# B&R Automation Studio project Embraco_LinkaNaOdlievanieRotorov_DokoncovaciaStanica_Rev2 (part 2)

#### Axis.c - Axis control
```c
 /********************************************************************
  * COPYRIGHT -- Bernecker + Rainer
  ********************************************************************
  * Author: Milan Jun
  * Created: May 28, 2014
  ********************************************************************/

#include <bur/plctypes.h>
#ifdef __cplusplus
	extern "C"
	{
#endif

#include "AxisLib.h"

#ifdef __cplusplus
	};
#endif

#define TRUE	1      /* Allways true */
#define FALSE 	0      /* Allways false */
#define DELAY   100    /* Delay time, it is dependence on cycle time */

/* Disabled all commands and executes */
void AxisDisableCmd (struct Axis* inst)
{

	/* RESET ALL FB EXECUTE/ENABLE INPUT */
	inst->internal.MC_Power_0.Enable = FALSE;
	inst->internal.MC_Home_0.Execute = FALSE;
	inst->internal.MC_Halt_0.Execute = FALSE;
	inst->internal.MC_Stop_0.Execute = FALSE;
	inst->internal.MC_MoveAbsolute_0.Execute = FALSE;
	inst->internal.MC_MoveAdditive_0.Execute = FALSE;
	inst->internal.MC_MoveVelocity_0.Execute = FALSE;
	inst->internal.MC_TorqueControl_0.Execute = FALSE;
	inst->internal.MC_BR_VelocityControl_0.Enable = FALSE;

	/* RESET USER COMMANDS */
	inst->cmd.home = FALSE;
	inst->cmd.halt = FALSE;
	inst->cmd.stop = FALSE;
	inst->cmd.moveAbsolute = FALSE;
	inst->cmd.moveAdditive = FALSE;
	inst->cmd.moveVelocity = FALSE;
	inst->cmd.moveVelocityControl = FALSE;
	inst->cmd.moveTorqueControl = FALSE;
	inst->cmd.moveJogPos = FALSE;
	inst->cmd.moveJogNeg = FALSE;
	inst->cmd.moveTorqueControl = FALSE;
	// inst->cmd.autoInicialization = FALSE;
	inst->errorID = FALSE;

}

/* Disabled all commands and executes */
void AxisAutoInicialization (struct Axis* inst)
{
 /* *************************************************************** *
 * ************** AUTO INICIALIZATION ENABLED ******************** *
 * *************************************************************** */
	switch (inst->internal.InitStep)
	{

		/* Init state */
		case STATE_INIT:
			inst->cmd.errorAck = FALSE;
			inst->internal.switch1 = FALSE;
			inst->internal.switch2 = FALSE;
			inst->internal.TimeCheck = 0;
			inst->internal.InitStep = STATE_WATCH;
			break;

		/* Wait for action, homing, power, error acknowledge */
		case STATE_WATCH:

			//   if ( (inst->status.DriveStatus.NetworkInit == TRUE) &&
			//   (inst->status.DriveStatus.HomingOk == FALSE) &&
			//   (inst->status.DriveStatus.ControllerStatus == TRUE) &&
			//   (inst->state.ErrorStop == FALSE) &&
			//			(inst->status.DriveStatus.AxisError == FALSE)	)
			//   {
			//    inst->internal.InitStep = STATE_HOME;
			//   }

			if ((inst->status.DriveStatus.NetworkInit == TRUE) &&
				(inst->status.DriveStatus.ControllerReady == TRUE) &&
				(inst->status.DriveStatus.ControllerStatus == FALSE) &&
				(inst->state.ErrorStop == FALSE) &&
				(inst->status.DriveStatus.AxisError == FALSE)	)
			{
				inst->internal.InitStep = STATE_SWITCHON;
			}

			if ((inst->status.DriveStatus.NetworkInit == TRUE) && ((inst->state.ErrorStop == TRUE) || (inst->status.DriveStatus.AxisError == TRUE) || (inst->errorID!=0)))
			{
				inst->internal.InitStep = STATE_ERROR_HANDLE;
			}
			break;

		/* State: homing */
		case STATE_HOME:

			if (inst->internal.switch1 == FALSE)
			{
				inst->cmd.home = TRUE;
				inst->internal.switch1 = TRUE;
			}

			if (inst->status.DriveStatus.HomingOk == TRUE)
			{
			inst->internal.InitStep = STATE_INIT;
			}

			inst->internal.TimeCheck = inst->internal.TimeCheck + 1;

			if (inst->internal.TimeCheck == DELAY)
			{
				inst->internal.InitStep = STATE_INIT;
				inst->internal.TimeCheck = 0;
			}
			break;

		/* State: switching on */
		case STATE_SWITCHON:

			if (inst->internal.switch1 == FALSE)
			{
				inst->cmd.power = TRUE;
				inst->internal.switch1 = TRUE;
			}

			if (inst->status.DriveStatus.ControllerStatus == TRUE)
			{
			inst->internal.InitStep = STATE_INIT;
			}

			inst->internal.TimeCheck = inst->internal.TimeCheck + 1;

			if (inst->internal.TimeCheck == DELAY)
			{
				inst->internal.InitStep = STATE_INIT;
				inst->internal.TimeCheck = 0;
			}
			break;

		/* State: automatic error acknowledge */
		case STATE_ERROR_HANDLE:

			inst->internal.errorOld = inst->errorID;

			if (inst->internal.switch1 == FALSE)
			{
			//inst->cmd.power = FALSE;
			inst->internal.switch1 = TRUE;
			}

			if ((inst->internal.switch1 == TRUE) && (inst->internal.switch2 == FALSE))
			{
			inst->cmd.errorAck = TRUE;
			inst->internal.switch2 = TRUE;
			}

			if (inst->internal.errorOld != inst->errorID)
			{
				inst->internal.errorOld = FALSE;
				inst->cmd.errorAck = FALSE;
				inst->internal.InitStep = STATE_INIT;
			}

			inst->internal.TimeCheck = inst->internal.TimeCheck + 1;

			if (inst->internal.TimeCheck == DELAY)
			{
				inst->internal.InitStep = STATE_INIT;
				inst->internal.TimeCheck = 0;
			}
			break;

	} /* END AutoInicialization enabled */

} /* END AutoInicialization disabled */

/* *************************************************************** *
 * ************************ AXIS CONTROL ************************* *
 * *************************************************************** */
void Axis(struct Axis* inst)
{

	/* Function Block is Enabled */
	if (inst->enable == TRUE){

		/* Function block active, when network iniciaization is true */
		if ( inst->status.DriveStatus.NetworkInit == TRUE )
		{
			inst->busy = FALSE;
			inst->active = TRUE;
		}
		else
		{
			inst->busy = TRUE;
			inst->active = FALSE;
		}

  /* *************************************************************** *
   * ************** AUTO INICIALIZATION DISABLED ******************* *
   * *************************************************************** */

		if ( inst->cmd.autoInicialization == FALSE )
		{
			inst->internal.switch1 = FALSE;
			inst->internal.TimeCheck = 0;
			inst->internal.InitStep = STATE_INIT;
		}
		else AxisAutoInicialization(inst);

  /* ******************** *
   * MC READ DRIVE STATUS *
   * ******************** */
		inst->internal.MC_BR_ReadDriveStatus_0.Enable = !inst->internal.MC_BR_ReadDriveStatus_0.Error;
		inst->internal.MC_BR_ReadDriveStatus_0.Axis = inst->par.axis;
		inst->internal.MC_BR_ReadDriveStatus_0.AdrDriveStatus = (UDINT)&inst->status.DriveStatus;

  /* ************** *
   * MC READ STATUS
   * ************** */
		inst->internal.MC_ReadStatus_0.Enable = !inst->internal.MC_ReadStatus_0.Error;
		inst->internal.MC_ReadStatus_0.Axis = inst->par.axis;

		/* MC READ ACTUAL POSITION */
		inst->internal.MC_ReadActualPosition_0.Enable = (!inst->internal.MC_ReadActualPosition_0.Error);
		inst->internal.MC_ReadActualPosition_0.Axis = inst->par.axis;

		if (inst->internal.MC_ReadActualPosition_0.Valid == TRUE)
		{
			inst->status.ActPosition = inst->internal.MC_ReadActualPosition_0.Position;
		}

		/* MC READ ACTUAL VELOCITY */
		inst->internal.MC_ReadActualVelocity_0.Enable = (!inst->internal.MC_ReadActualVelocity_0.Error);
		inst->internal.MC_ReadActualVelocity_0.Axis = inst->par.axis;

		if(inst->internal.MC_ReadActualVelocity_0.Valid == TRUE)
		{
			inst->status.ActVelocity = inst->internal.MC_ReadActualVelocity_0.Velocity;
		}

		/* MC READ ACTUAL TORQUE */
		inst->internal.MC_ReadActualTorque_0.Enable = (!inst->internal.MC_ReadActualTorque_0.Error);
		inst->internal.MC_ReadActualTorque_0.Axis = inst->par.axis;

		if(inst->internal.MC_ReadActualTorque_0.Valid == TRUE)
		{
			inst->status.ActTorque = inst->internal.MC_ReadActualTorque_0.Torque;
		}

		/* MC READ AXIS ERROR */
		inst->internal.MC_ReadAxisError_0.Enable = !inst->internal.MC_ReadAxisError_0.Error;
		inst->internal.MC_ReadAxisError_0.Axis = inst->par.axis;
		inst->internal.MC_ReadAxisError_0.DataAddress = (UDINT)&(inst->errorText);
		inst->internal.MC_ReadAxisError_0.DataLength = sizeof(inst->errorText);
		brsstrcpy((void*)&inst->internal.MC_ReadAxisError_0.DataObjectName, "acp10etxen");

		/* CHECK FOR GENERAL AXIS ERROR */
		if ((inst->internal.MC_ReadAxisError_0.AxisErrorID != FALSE) &&
			(inst->internal.MC_ReadAxisError_0.Valid == TRUE))
		{
			inst->internal.AxisStep = AXISSTATE_ERROR_AXIS;
		}

		/* Main Cyclic Part */

		if ( inst->cmd.power == FALSE )
		{
			inst->internal.MC_Power_0.Enable = FALSE;
			inst->internal.AxisStep = AXISSTATE_WAIT;
		}

		/* State machine for axis */
		switch (inst->internal.AxisStep)
		{
			/* STATE WAIT FOR POWERON */
			case AXISSTATE_WAIT:

				/* WAIT FOR POWERON COMMAND */
				if (inst->cmd.power == TRUE) {
					inst->internal.AxisStep = AXISSTATE_POWER_ON;
				}
				else {
					inst->internal.MC_Power_0.Enable = FALSE;
				}

				AxisDisableCmd(inst);

				break;

   /* *************************************************************** *
    * ************************ STATE POWER ON *********************** *
    * *************************************************************** */
			case AXISSTATE_POWER_ON:
				inst->internal.MC_Power_0.Axis = inst->par.axis;
				inst->internal.MC_Power_0.Enable = TRUE;

				/* Check staus ok */
				if (inst->internal.MC_Power_0.Status == TRUE) {
					inst->internal.AxisStep = AXISSTATE_READY;
				}
				/* Check a power error, then go to error state */
				if (inst->internal.MC_Power_0.Error == TRUE) {
					inst->errorID = inst->internal.MC_Power_0.ErrorID;
					inst->internal.AxisStep = AXISSTATE_ERROR;
				}
				break;
			/* ************************************************************** */

			/* ************************************************************** *
			* ************************* STATE READY ************************* *
			* *************************************************************** */
			case AXISSTATE_READY:
				if (inst->cmd.home == TRUE) {
					inst->internal.AxisStep = AXISSTATE_HOME;
				}

				else if (inst->cmd.stop == TRUE) {
					inst->cmd.stop = FALSE;
					inst->internal.AxisStep = AXISSTATE_STOP;
				}
					else if (inst->cmd.moveAbsolute == TRUE) {
						inst->cmd.moveAbsolute = FALSE;
						inst->internal.AxisStep = AXISSTATE_MOVE_ABSOLUTE;
					}
						else if (inst->cmd.moveAdditive == TRUE) {
							inst->cmd.moveAdditive = FALSE;
							inst->internal.AxisStep = AXISSTATE_MOVE_ADDITIVE;
						}
							else if (inst->cmd.moveVelocity == TRUE && inst->par.blockMoveVelocity == FALSE) {
								inst->cmd.moveVelocity = FALSE;
								inst->internal.AxisStep = AXISSTATE_MOVE_VELOCITY;
							}
								else if (inst->cmd.moveJogPos == TRUE) {
									inst->cmd.moveVelocity = FALSE;
									inst->internal.AxisStep = AXISSTATE_MOVE_JOGPOS;
								}
									else if (inst->cmd.moveJogNeg == TRUE) {
										inst->cmd.moveVelocity = FALSE;
										inst->internal.AxisStep = AXISSTATE_MOVE_JOGNEG;
									}
										else if (inst->cmd.moveTorqueControl == TRUE) {
											inst->cmd.moveTorqueControl = FALSE;
											inst->internal.AxisStep = AXISSTATE_MOVE_TORQUE_CONTROL;
										}
											else if (inst->cmd.moveVelocityControl == TRUE) {
												inst->cmd.moveVelocityControl = FALSE;
												inst->internal.AxisStep = AXISSTATE_MOVE_VELOCITY_CONTROL;
											}
												else if (inst->cmd.halt == TRUE) {
													inst->cmd.halt = FALSE;
													inst->internal.AxisStep = AXISSTATE_HALT;
												}
				break;

   /* ************************************************************** *
   * ************************** STATE HOME ************************* *
   * *************************************************************** */
			case AXISSTATE_HOME:
				inst->internal.MC_Home_0.Axis = inst->par.axis;
				inst->internal.MC_Home_0.Position = inst->par.homePos;
				inst->internal.MC_Home_0.HomingMode = inst->par.homeMode;
				inst->internal.MC_Home_0.Execute = TRUE;

				/* Check status done */
				if (inst->internal.MC_Home_0.Done == TRUE) {
					inst->cmd.home = FALSE;
					inst->internal.MC_Home_0.Execute = FALSE;
					inst->internal.AxisStep = AXISSTATE_READY;
				}

				/*Check command stop*/
				if (inst->cmd.stop == TRUE) {
					inst->cmd.home = FALSE;
					inst->cmd.stop = FALSE;
					inst->internal.MC_Home_0.Execute = FALSE;
					inst->internal.AxisStep = AXISSTATE_STOP;
				}

				/* Check a homing error, then go to error state */
				if (inst->internal.MC_Home_0.Error == TRUE) {
					inst->internal.MC_Home_0.Execute = FALSE;
					inst->errorID = inst->internal.MC_Home_0.ErrorID;
					inst->internal.AxisStep = AXISSTATE_ERROR;
				}
				break;

   /* ************************************************************** *
   * ************************** STATE HALT ************************* *
   * *************************************************************** */
			case AXISSTATE_HALT:
				inst->internal.MC_Halt_0.Axis = inst->par.axis;
				inst->internal.MC_Halt_0.Deceleration = inst->par.dec;
				inst->internal.MC_Halt_0.Execute = TRUE;

				/* Check status done */
				if (inst->internal.MC_Halt_0.Done == TRUE) {
					inst->internal.MC_Halt_0.Execute = FALSE;
					inst->internal.AxisStep = AXISSTATE_READY;
				}
				/* Check status command aborted */
				else if (inst->internal.MC_Halt_0.CommandAborted == TRUE) {
					inst->internal.MC_Halt_0.Execute = FALSE;
					inst->internal.AxisStep = AXISSTATE_HALT;
				}
				/* Check a halt error, then go to error state */
				if (inst->internal.MC_Halt_0.Error == TRUE) {
					inst->internal.MC_Halt_0.Execute = FALSE;
					inst->errorID = inst->internal.MC_Home_0.ErrorID;
					inst->internal.AxisStep = AXISSTATE_ERROR;
				}
				break;

   /* ************************************************************** *
   * ************************** STATE STOP ************************* *
   * *************************************************************** */
			case AXISSTATE_STOP:
				inst->internal.MC_Stop_0.Axis = inst->par.axis;
				inst->internal.MC_Stop_0.Deceleration = inst->par.dec;
				inst->internal.MC_Stop_0.Execute = TRUE;

				/* Check status ok */
				if ((inst->internal.MC_Stop_0.Done == TRUE) && (inst->cmd.stop == FALSE))
				{
					inst->internal.MC_Stop_0.Execute = FALSE;
					inst->internal.AxisStep = AXISSTATE_READY;
				}
				/* Check status command aborted */
				else if (inst->internal.MC_Stop_0.CommandAborted == TRUE) {
					inst->internal.MC_Stop_0.Execute = FALSE;
					inst->internal.AxisStep = AXISSTATE_STOP;
				}
				/* Check a stop error, then go to error state */
				if (inst->internal.MC_Stop_0.Error == TRUE)
				{
					inst->internal.MC_Stop_0.Execute = FALSE;
					inst->errorID = inst->internal.MC_Stop_0.ErrorID;
					inst->internal.AxisStep = AXISSTATE_ERROR;
				}
				break;

   /* ************************************************************** *
   * ********************** STATE MOVE ABSOLUTE ******************** *
   * *************************************************************** */
			case AXISSTATE_MOVE_ABSOLUTE:
				inst->internal.MC_MoveAbsolute_0.Axis = inst->par.axis;
				inst->internal.MC_MoveAbsolute_0.Position = inst->par.position;
				inst->internal.MC_MoveAbsolute_0.Velocity = inst->par.velocity;
				inst->internal.MC_MoveAbsolute_0.Acceleration = inst->par.acc;
				inst->internal.MC_MoveAbsolute_0.Deceleration = inst->par.dec;
				inst->internal.MC_MoveAbsolute_0.Direction = inst->par.direction;
				inst->internal.MC_MoveAbsolute_0.Execute = TRUE;

				/* Check status done */
				if (inst->internal.MC_MoveAbsolute_0.Done == TRUE) {
					inst->internal.MC_MoveAbsolute_0.Execute = FALSE;
					inst->internal.AxisStep = AXISSTATE_READY;
				}

				/* Check command halt */
				if	(inst->cmd.halt == TRUE) {
					inst->cmd.moveAbsolute = FALSE;
					inst->cmd.halt = FALSE;
					inst->internal.MC_MoveAbsolute_0.Execute = FALSE;
					inst->internal.AxisStep = AXISSTATE_HALT;
				}

				/*Check command stop*/
				if (inst->cmd.stop == TRUE) {
					inst->cmd.moveAbsolute = FALSE;
					inst->cmd.stop = FALSE;
					inst->internal.MC_MoveAbsolute_0.Execute = FALSE;
					inst->internal.AxisStep = AXISSTATE_STOP;
				}

				/* Check a halt error, then go to error state */
				if (inst->internal.MC_MoveAbsolute_0.Error == TRUE)
				{
					inst->internal.MC_MoveAbsolute_0.Execute = FALSE;
					inst->errorID = inst->internal.MC_MoveAbsolute_0.ErrorID;
					inst->internal.AxisStep = AXISSTATE_ERROR;
				}
				break;

   /* ************************************************************** *
   * ********************** STATE MOVE ADDITIVE ******************** *
   * *************************************************************** */
			case AXISSTATE_MOVE_ADDITIVE:
				inst->internal.MC_MoveAdditive_0.Axis = inst->par.axis;
				inst->internal.MC_MoveAdditive_0.Velocity = inst->par.velocity;
				inst->internal.MC_MoveAdditive_0.Distance = inst->par.distance;
				inst->internal.MC_MoveAdditive_0.Acceleration = inst->par.acc;
				inst->internal.MC_MoveAdditive_0.Deceleration = inst->par.dec;
				inst->internal.MC_MoveAdditive_0.Execute = TRUE;

				/*Check command stop*/
				if (inst->cmd.stop == TRUE) {
					inst->cmd.moveAdditive = FALSE;
					inst->cmd.stop = FALSE;
					inst->internal.MC_MoveAdditive_0.Execute = FALSE;
					inst->internal.AxisStep = AXISSTATE_STOP;
				}

				/* Check status ok */
				if (inst->cmd.halt == TRUE)
				{
					inst->cmd.halt = FALSE;
					inst->internal.MC_MoveAdditive_0.Execute = FALSE;
					inst->internal.AxisStep = AXISSTATE_HALT;
				}
				else if (inst->internal.MC_MoveAdditive_0.Done == TRUE)
				{
					inst->internal.MC_MoveAdditive_0.Execute = FALSE;
					inst->internal.AxisStep = AXISSTATE_READY;
				}
				/* Check a halt error, then go to error state */
				if (inst->internal.MC_MoveAdditive_0.Error == TRUE)
				{
					inst->internal.MC_MoveAdditive_0.Execute = FALSE;
					inst->errorID = inst->internal.MC_MoveAdditive_0.ErrorID;
					inst->internal.AxisStep = AXISSTATE_ERROR;
				}
				break;

			/* State move velocity */
			case AXISSTATE_MOVE_VELOCITY:
				inst->internal.MC_MoveVelocity_0.Axis = inst->par.axis;
				inst->internal.MC_MoveVelocity_0.Velocity = inst->par.velocity;
				inst->internal.MC_MoveVelocity_0.Acceleration = inst->par.acc;
				inst->internal.MC_MoveVelocity_0.Deceleration = inst->par.dec;
				inst->internal.MC_MoveVelocity_0.Direction = inst->par.direction;
				inst->internal.MC_MoveVelocity_0.Execute = TRUE;

				/*Check command stop*/
				if (inst->cmd.stop == TRUE) {
					inst->cmd.moveVelocity = FALSE;
					inst->cmd.stop = FALSE;
					inst->internal.MC_MoveVelocity_0.Execute = FALSE;
					inst->internal.AxisStep = AXISSTATE_STOP;
				}

				/* check if commanded halt is reached */
				if	(inst->cmd.halt == TRUE)
				{
					inst->cmd.halt = FALSE;
					inst->internal.MC_MoveVelocity_0.Execute = FALSE;
					inst->internal.AxisStep = AXISSTATE_HALT;
				}
				/* check if commanded invelocity is reached */
				else if (inst->internal.MC_MoveVelocity_0.InVelocity == TRUE)
				{
					inst->internal.MC_MoveVelocity_0.Execute = FALSE;
					inst->internal.AxisStep = AXISSTATE_READY;
				}
					else if (inst->par.blockMoveVelocity == TRUE)
					{
						inst->internal.MC_MoveVelocity_0.Execute = FALSE;
						inst->internal.AxisStep = AXISSTATE_HALT;
					}

				/* Check a halt error, then go to error state */
				if (inst->internal.MC_MoveVelocity_0.Error == TRUE)
				{
					inst->internal.MC_MoveVelocity_0.Execute = FALSE;
					inst->errorID = inst->internal.MC_MoveVelocity_0.ErrorID;
					inst->internal.AxisStep = AXISSTATE_ERROR;
				}
				break;

			/* State move jog positive */
			case AXISSTATE_MOVE_JOGPOS:
				inst->internal.MC_MoveVelocity_0.Axis = inst->par.axis;
				inst->internal.MC_MoveVelocity_0.Velocity = inst->par.velocityJog;
				inst->internal.MC_MoveVelocity_0.Acceleration = inst->par.acc;
				inst->internal.MC_MoveVelocity_0.Deceleration = inst->par.dec;
				inst->internal.MC_MoveVelocity_0.Direction = mcPOSITIVE_DIR;
				inst->internal.MC_MoveVelocity_0.Execute = TRUE;

				/* check if commanded velocity */
				if	(inst->cmd.moveJogPos == FALSE) {
					inst->internal.MC_MoveVelocity_0.Execute = FALSE;
					inst->internal.AxisStep = AXISSTATE_HALT;
				}

				/* Check a halt error, then go to error state */
				if (inst->internal.MC_MoveVelocity_0.Error == TRUE) {
					inst->internal.MC_MoveVelocity_0.Execute = FALSE;
					inst->errorID = inst->internal.MC_MoveVelocity_0.ErrorID;
					inst->internal.AxisStep = AXISSTATE_ERROR;
				}
				break;

			/* State move jog negative */
			case AXISSTATE_MOVE_JOGNEG:
				inst->internal.MC_MoveVelocity_0.Axis = inst->par.axis;
				inst->internal.MC_MoveVelocity_0.Velocity = inst->par.velocityJog;
				inst->internal.MC_MoveVelocity_0.Acceleration = inst->par.acc;
				inst->internal.MC_MoveVelocity_0.Deceleration = inst->par.dec;
				inst->internal.MC_MoveVelocity_0.Direction = mcNEGATIVE_DIR;
				inst->internal.MC_MoveVelocity_0.Execute = TRUE;

				/* check if commanded velocity */
				if	(inst->cmd.moveJogNeg == FALSE)
				{
					inst->internal.MC_MoveVelocity_0.Execute = FALSE;
					inst->internal.AxisStep = AXISSTATE_HALT;
				}

				/* Check a halt error, then go to error state */
				if (inst->internal.MC_MoveVelocity_0.Error == TRUE)
				{
					inst->internal.MC_MoveVelocity_0.Execute = FALSE;
					inst->errorID = inst->internal.MC_MoveVelocity_0.ErrorID;
					inst->internal.AxisStep = AXISSTATE_ERROR;
				}
				break;

			/* State move torque control */
			case AXISSTATE_MOVE_TORQUE_CONTROL:

				inst->internal.MC_TorqueControl_0.Axis = inst->par.axis;
				inst->internal.MC_TorqueControl_0.Torque = inst->par.torque;
				inst->internal.MC_TorqueControl_0.TorqueRamp = inst->par.torqueRamp;
				inst->internal.MC_TorqueControl_0.Velocity = inst->par.velocity;
				inst->internal.MC_TorqueControl_0.Acceleration = inst->par.acc;
				inst->internal.MC_TorqueControl_0.Execute = TRUE;

				/*Check command stop*/
				if (inst->cmd.stop == TRUE) {
					inst->cmd.moveTorqueControl = FALSE;
					inst->cmd.stop = FALSE;
					inst->internal.MC_TorqueControl_0.Execute = FALSE;
					inst->internal.AxisStep = AXISSTATE_STOP;
				}

				/* check if commanded halt is reached */
				if	(inst->cmd.halt == TRUE)
				{
					inst->cmd.halt = FALSE;
					inst->internal.MC_TorqueControl_0.Execute = FALSE;
					inst->internal.AxisStep = AXISSTATE_HALT;
				}

				/* Check a halt error, then go to error state */
				if (inst->internal.MC_TorqueControl_0.Error == TRUE)
				{
					inst->internal.MC_TorqueControl_0.Execute = FALSE;
					inst->errorID = inst->internal.MC_TorqueControl_0.ErrorID;
					inst->internal.AxisStep = AXISSTATE_ERROR;
				}
				break;

			case AXISSTATE_MOVE_VELOCITY_CONTROL:
				inst->internal.MC_BR_VelocityControl_0.Axis = inst->par.axis;
				inst->internal.MC_BR_VelocityControl_0.CyclicVelocity = inst->par.velocityControl.cyclicVelocity;
				inst->internal.MC_BR_VelocityControl_0.CyclicVelocityCorrection = inst->par.velocityControl.cyclicVelocityCorrection;
				inst->internal.MC_BR_VelocityControl_0.CyclicTorque = inst->par.velocityControl.cyclicTorque;
				inst->internal.MC_BR_VelocityControl_0.TorqueMode = inst->par.velocityControl.TorqueMode;
				inst->internal.MC_BR_VelocityControl_0.Acceleration = inst->par.acc;
				inst->internal.MC_BR_VelocityControl_0.Deceleration = inst->par.dec;
				inst->internal.MC_BR_VelocityControl_0.SctrlKv = inst->par.velocityControl.sCtrlKv;
				inst->internal.MC_BR_VelocityControl_0.SctrlTn = inst->par.velocityControl.sCtrlTn;
				inst->internal.MC_BR_VelocityControl_0.InitSctrl = inst->par.velocityControl.initSctrl;
				inst->internal.MC_BR_VelocityControl_0.Enable = TRUE;

				/* check if commanded halt */
				if	(inst->cmd.halt == TRUE)
				{
					inst->cmd.halt = FALSE;
					inst->internal.MC_BR_VelocityControl_0.Enable = FALSE;
					inst->internal.AxisStep = AXISSTATE_READY;
				}

				/*Check command stop*/
				if (inst->cmd.stop == TRUE) {
					inst->cmd.moveVelocityControl = FALSE;
					inst->cmd.stop = FALSE;
					inst->internal.MC_BR_VelocityControl_0.Enable = FALSE;
					inst->internal.AxisStep = AXISSTATE_STOP;
				}

				/* Check a halt error, then go to error state */
				if (inst->internal.MC_BR_VelocityControl_0.Error == TRUE)
				{
					inst->internal.MC_BR_VelocityControl_0.Enable = FALSE;
					inst->errorID = inst->internal.MC_BR_VelocityControl_0.ErrorID;
					inst->internal.AxisStep = AXISSTATE_ERROR;
				}
				break;

			/* State axis error */
			case AXISSTATE_ERROR:
				inst->errorCount++;
				inst->error = TRUE;
				/* check if FB indicates an axis error */
				if (inst->internal.MC_ReadAxisError_0.AxisErrorCount != FALSE) {
					inst->internal.AxisStep = AXISSTATE_ERROR_AXIS;
				}
				else {
					if (inst->cmd.errorAck == TRUE) {
						inst->cmd.errorAck = FALSE;
						inst->errorID = 0;

						/* reset axis if it is in axis state ErrorStop */
						if ((inst->internal.MC_ReadStatus_0.Errorstop == TRUE) && (inst->internal.MC_ReadStatus_0.Valid == TRUE)) {
							inst->internal.AxisStep = AXISSTATE_ERROR_RESET;
						}
						else {
							inst->error = FALSE;
							inst->internal.AxisStep = AXISSTATE_WAIT;
						}
					}
				}
				break;

			/* State error axis */
			case AXISSTATE_ERROR_AXIS:
				inst->errorID = TRUE;
				if (inst->internal.MC_ReadAxisError_0.Valid == TRUE)
				{
					if (inst->internal.MC_ReadAxisError_0.AxisErrorID != FALSE)
					{
						inst->errorID = inst->internal.MC_ReadAxisError_0.AxisErrorID;
					}
					inst->internal.MC_ReadAxisError_0.Acknowledge = FALSE;
					if (inst->cmd.errorAck == TRUE)
					{
						inst->cmd.errorAck = FALSE;
						/* acknowledge axis error */
						if (inst->internal.MC_ReadAxisError_0.AxisErrorID != FALSE)
						{
							inst->internal.MC_ReadAxisError_0.Acknowledge = TRUE;
						}
					}
					if (inst->internal.MC_ReadAxisError_0.AxisErrorCount == FALSE)
					{
						inst->errorID = FALSE;
						/* reset axis if it is in axis state ErrorStop */
						if ((inst->internal.MC_ReadStatus_0.Errorstop == 1) && (inst->internal.MC_ReadStatus_0.Valid == 1))
						{
							inst->internal.AxisStep = AXISSTATE_ERROR_RESET;
						}
						else
						{
							inst->error = FALSE;
							inst->internal.AxisStep = AXISSTATE_WAIT;
						}
					}
				}
				break;

			/* State error reset */
			case AXISSTATE_ERROR_RESET:

				inst->internal.MC_Reset_0.Axis = inst->par.axis;
				inst->internal.MC_Reset_0.Execute = TRUE;

				/* reset MC_Power.Enable if this FB is in Error*/
				if (inst->internal.MC_Power_0.Error == TRUE)
				{
					inst->internal.MC_Power_0.Enable = FALSE;
				}
				if (inst->internal.MC_Reset_0.Done == TRUE)
				{
					inst->internal.MC_Reset_0.Execute = FALSE;
					inst->error = FALSE;
					inst->internal.AxisStep = AXISSTATE_WAIT;
				}
				else if (inst->internal.MC_Reset_0.Error == TRUE)
				{
					inst->internal.MC_Reset_0.Execute = FALSE;
					inst->internal.AxisStep = AXISSTATE_ERROR;
				}
				break;
		}

	} /* Main End */

	/* Function block is Disabled */
	else {

		inst->active = FALSE;
		inst->busy = FALSE;

		inst->cmd.power = FALSE;
		AxisDisableCmd(inst);
	}

	if (inst->internal.MC_ReadStatus_0.Valid == TRUE) {
		inst->state.Disabled = inst->internal.MC_ReadStatus_0.Disabled;
		inst->state.StandStill = inst->internal.MC_ReadStatus_0.StandStill;
		inst->state.Stopping = inst->internal.MC_ReadStatus_0.Stopping;
		inst->state.Homing = inst->internal.MC_ReadStatus_0.Homing;
		inst->state.DiscreteMotion = inst->internal.MC_ReadStatus_0.DiscreteMotion;
		inst->state.ContinuousMotion = inst->internal.MC_ReadStatus_0.ContinuousMotion;
		inst->state.SynchronizedMotion = inst->internal.MC_ReadStatus_0.SynchronizedMotion;
		inst->state.ErrorStop = inst->internal.MC_ReadStatus_0.Errorstop;
	}
	else {
		inst->state.Disabled = FALSE;
		inst->state.StandStill = FALSE;
		inst->state.Stopping = FALSE;
		inst->state.Homing = FALSE;
		inst->state.DiscreteMotion = FALSE;
		inst->state.ContinuousMotion = FALSE;
		inst->state.SynchronizedMotion = FALSE;
		inst->state.ErrorStop = FALSE;
	}

	MC_BR_ReadDriveStatus(&inst->internal.MC_BR_ReadDriveStatus_0);
	MC_ReadStatus(&inst->internal.MC_ReadStatus_0);
	MC_ReadActualPosition(&inst->internal.MC_ReadActualPosition_0);
	MC_ReadActualVelocity(&inst->internal.MC_ReadActualVelocity_0);
	MC_ReadActualTorque(&inst->internal.MC_ReadActualTorque_0);
	MC_ReadAxisError(&inst->internal.MC_ReadAxisError_0);
	MC_Reset(&inst->internal.MC_Reset_0);
	MC_Power(&inst->internal.MC_Power_0);
	MC_Home(&inst->internal.MC_Home_0);
	MC_Halt(&inst->internal.MC_Halt_0);
	MC_Stop(&inst->internal.MC_Stop_0);
	MC_MoveAbsolute(&inst->internal.MC_MoveAbsolute_0);
	MC_MoveAdditive(&inst->internal.MC_MoveAdditive_0);
	MC_MoveVelocity(&inst->internal.MC_MoveVelocity_0);
	MC_TorqueControl(&inst->internal.MC_TorqueControl_0);
	MC_BR_VelocityControl(&inst->internal.MC_BR_VelocityControl_0);

}
```

#### AxisExtension.c - Axis extension control/status
```c
#include <bur/plctypes.h>
#ifdef __cplusplus
	extern "C"
	{
#endif
	#include "AxisLib.h"
#ifdef __cplusplus
	};
#endif

#define TRUE		  1      /* Allways true */
#define FALSE 		0      /* Allways false */
#define DELAY   100    /* Delay time, it is dependence on cycle time */

void AxisExtension(struct AxisExtension* inst)
{

   /* *************************************************************** *
   * ******************* READ / WRITE PARID ************************ *
   * *************************************************************** */

 unsigned long int encoderResetValue = 1;
 unsigned short int brakeMode = 0;

 if (inst->enable == FALSE)
 {
  inst->internal.AxisReadStep = 0;
		inst->active = FALSE;
 }

 else
		inst->active = TRUE;
 {
  switch (inst->internal.AxisReadStep)
  {

   /* Wait for command */
   case 0:

    /* 719: Encoder1: Encoder command */
    if (inst->cmd.cmdRstEncoder == TRUE)
    {
     inst->cmd.cmdRstEncoder = FALSE;
     inst->internal.AxisReadStep = 1;
    }
    /* Command unbrake */
    else if ( inst->cmd.cmdUnbrake == TRUE )
    {
     inst->internal.AxisReadStep = 2;
     inst->cmd.cmdUnbrake = FALSE;
    }
    /* Command brake */
    else if ( inst->cmd.cmdBrake == TRUE )
    {
     inst->internal.AxisReadStep = 3;
     inst->cmd.cmdBrake = FALSE;
    }
    /* Command toggle brake/unbrake */
    else if ( inst->cmd.cmdBrakeToggle == TRUE )
    {
     inst->internal.AxisReadStep = 4;
     inst->cmd.cmdBrakeToggle = FALSE;
    }
					/* Command for reading hardware info */
				else if ( inst->cmd.cmdGetHwInfo == TRUE )
				{
					inst->internal.AxisReadStep = 5;
					inst->cmd.cmdGetHwInfo = FALSE;
				}
				/* Continue with reading parid */
				else {
					inst->internal.AxisReadStep = 10;
				}
    break;

   /* Reset encoder */
   case 1:

    inst->internal.MC_BR_WriteParID_0.Execute = 1;
    inst->internal.MC_BR_WriteParID_0.Axis = inst->par.axis;
    inst->internal.MC_BR_WriteParID_0.ParID = 719;
    inst->internal.MC_BR_WriteParID_0.DataAddress = (UDINT)&(encoderResetValue);
    inst->internal.MC_BR_WriteParID_0.DataType = ncPAR_TYP_UDINT;

    if (inst->internal.MC_BR_WriteParID_0.Done == TRUE)
    {
     inst->internal.MC_BR_WriteParID_0.Execute = FALSE;
     inst->internal.AxisReadStep = 0;
    }
    else if (inst->internal.MC_BR_WriteParID_0.Busy == TRUE)
    {
     /* busy */
    }
    if (inst->internal.MC_BR_WriteParID_0.Error == TRUE)
    {
     inst->internal.MC_BR_WriteParID_0.Execute = FALSE;
     inst->internal.AxisReadStep = 0;
    }
    break;

   /* Brake operation */
   case 2:
    inst->internal.MC_BR_BrakeOperation_0.Execute = TRUE;
    inst->internal.MC_BR_BrakeOperation_0.Axis = inst->par.axis;
    inst->internal.MC_BR_BrakeOperation_0.BrakeCommand = 1;

    if (inst->internal.MC_BR_BrakeOperation_0.Done == TRUE)
    {
     inst->internal.MC_BR_BrakeOperation_0.Execute = FALSE;
     inst->internal.AxisReadStep = 0;
    }
    else if (inst->internal.MC_BR_BrakeOperation_0.Busy == TRUE)
    {
     /* busy */
    }

    /* Check a error, then go to error state */
    if (inst->internal.MC_BR_BrakeOperation_0.Error == TRUE)
    {
     inst->internal.MC_BR_BrakeOperation_0.Execute = FALSE;
     inst->errorID = inst->internal.MC_BR_BrakeOperation_0.ErrorID;
     inst->internal.AxisReadStep = 0;
    }
    break;

   /* unBrake operation */
   case 3:
    inst->internal.MC_BR_BrakeOperation_0.Execute = TRUE;
    inst->internal.MC_BR_BrakeOperation_0.Axis = inst->par.axis;
    inst->internal.MC_BR_BrakeOperation_0.BrakeCommand = 0;

    if (inst->internal.MC_BR_BrakeOperation_0.Done == TRUE)
    {
     inst->internal.MC_BR_BrakeOperation_0.Execute = FALSE;
     inst->internal.AxisReadStep = 0;
    }
    else if (inst->internal.MC_BR_BrakeOperation_0.Busy == TRUE)
    {
     /* busy */
    }

    /* Check a error, then go to error state */
    if (inst->internal.MC_BR_BrakeOperation_0.Error == TRUE)
    {
     inst->internal.MC_BR_BrakeOperation_0.Execute = FALSE;
     inst->errorID = inst->internal.MC_BR_BrakeOperation_0.ErrorID;
     inst->internal.AxisReadStep = 0;
    }
    break;

   /* unBrake operation */
   case 4:
    inst->internal.MC_BR_BrakeOperation_0.Execute = TRUE;
    inst->internal.MC_BR_BrakeOperation_0.Axis = inst->par.axis;
    inst->internal.MC_BR_BrakeOperation_0.BrakeCommand = inst->internal.brakeMode;

    if (inst->internal.MC_BR_BrakeOperation_0.Done == TRUE)
    {
     inst->internal.brakeMode = !inst->internal.brakeMode;
     inst->internal.MC_BR_BrakeOperation_0.Execute = FALSE;
     inst->internal.AxisReadStep = 0;
    }
    else if (inst->internal.MC_BR_BrakeOperation_0.Busy == TRUE)
    {
     /* busy */
    }

    /* Check a error, then go to error state */
    if (inst->internal.MC_BR_BrakeOperation_0.Error == TRUE)
    {
     inst->internal.MC_BR_BrakeOperation_0.Execute = FALSE;
     inst->errorID = inst->internal.MC_BR_BrakeOperation_0.ErrorID;
     inst->internal.AxisReadStep = 0;
    }
    break;

			/* Get hardware information */
			case 5:
				inst->internal.MC_BR_GetHardwareInfo_0.Execute = TRUE;
				inst->internal.MC_BR_GetHardwareInfo_0.Axis = inst->par.axis;

				brsmemset( &(inst->internal.MC_BR_GetHardwareInfo_0.HardwareInfo),0,sizeof(inst->internal.MC_BR_GetHardwareInfo_0.HardwareInfo));

				if (inst->internal.MC_BR_GetHardwareInfo_0.Done == TRUE)
				{
					inst->internal.MC_BR_GetHardwareInfo_0.Execute = FALSE;
				 inst->status.HardwareInfo = inst->internal.MC_BR_GetHardwareInfo_0.HardwareInfo;

				 brsmemcpy( &(inst->internal.MC_BR_GetHardwareInfo_0.HardwareInfo), &(inst->internal.MC_BR_GetHardwareInfo_0.HardwareInfo),sizeof(inst->internal.MC_BR_GetHardwareInfo_0.HardwareInfo));

					inst->internal.AxisReadStep = 0;
				}
				else if (inst->internal.MC_BR_GetHardwareInfo_0.Busy == TRUE)
				{
					/* busy */
				}

				/* Check a error, then go to error state */
				if (inst->internal.MC_BR_GetHardwareInfo_0.Error == TRUE)
				{
					inst->internal.MC_BR_GetHardwareInfo_0.Execute = FALSE;
					inst->errorID = inst->internal.MC_BR_GetHardwareInfo_0.ErrorID;
					inst->internal.AxisReadStep = 0;
				}
				break;

   /* Continue with reading temperature */
   case 10:
				if ( inst->cmd.cmdReadTemp == TRUE ){

					inst->internal.MC_BR_ReadParID_0.Execute = 1;
					inst->internal.MC_BR_ReadParID_0.Axis = inst->par.axis;
					inst->internal.MC_BR_ReadParID_0.ParID = 381; /* 381: Temperature sensor: Temperature | TEMP_MOTOR | RD | °C | REAL */
					inst->internal.MC_BR_ReadParID_0.DataAddress = (UDINT)&(inst->status.ActMotorTemp);
					inst->internal.MC_BR_ReadParID_0.DataType = ncPAR_TYP_REAL;

					if (inst->internal.MC_BR_ReadParID_0.Done == TRUE)
					{
						inst->internal.MC_BR_ReadParID_0.Execute = FALSE;
						inst->internal.AxisReadStep++;
					}
					else if (inst->internal.MC_BR_ReadParID_0.Busy == TRUE) { }

				 /* If mc_br_readparid error */
					if (inst->internal.MC_BR_ReadParID_0.Error == TRUE)
					{
						inst->internal.MC_BR_ReadParID_0.Execute = FALSE;
						inst->internal.AxisReadStep = 0;
					}
				}
				else {
					inst->internal.AxisReadStep++;
					inst->status.ActMotorTemp = 0;
				}
    break;

			/* Continue with reading current */
   case 11:
				if ( inst->cmd.cmdReadCurrent == TRUE ) {
					inst->internal.MC_BR_ReadParID_0.Execute = 1;
					inst->internal.MC_BR_ReadParID_0.Axis = inst->par.axis;
					inst->internal.MC_BR_ReadParID_0.ParID = 214; /* 214: CTRL Current controller: Actual stator current quadrature component | ICTRL_ISQ_ACT | RD | A | REAL */
					inst->internal.MC_BR_ReadParID_0.DataAddress = (UDINT)&(inst->status.ActMotorCurrent);
					inst->internal.MC_BR_ReadParID_0.DataType = ncPAR_TYP_REAL ;

					if (inst->internal.MC_BR_ReadParID_0.Done == TRUE)
					{
						inst->internal.MC_BR_ReadParID_0.Execute = FALSE;
						inst->internal.AxisReadStep++;
					}
					else if (inst->internal.MC_BR_ReadParID_0.Busy == TRUE){ }

				 /* If mc_br_readparid error */
					if (inst->internal.MC_BR_ReadParID_0.Error == TRUE)
					{
						inst->internal.MC_BR_ReadParID_0.Execute = FALSE;
						inst->internal.AxisReadStep = 0;
					}
				}
				else {
					inst->internal.AxisReadStep++;
					inst->status.ActMotorCurrent = 0;
				}
    break;

			/* Continue with reading lag error */
   case 12:
				if ( inst->cmd.cmdReadLagError == TRUE ) {
					inst->internal.MC_BR_ReadParID_0.Execute = 1;
					inst->internal.MC_BR_ReadParID_0.Axis = inst->par.axis;
					inst->internal.MC_BR_ReadParID_0.ParID = 112; /* 112: CTRL Position controller: Lag error */
					inst->internal.MC_BR_ReadParID_0.DataAddress = (UDINT)&(inst->status.ActLagError);
					inst->internal.MC_BR_ReadParID_0.DataType = ncPAR_TYP_REAL ;

					if (inst->internal.MC_BR_ReadParID_0.Done == TRUE)
					{
						inst->internal.MC_BR_ReadParID_0.Execute = FALSE;
						inst->internal.AxisReadStep = 0;
					}
					else if (inst->internal.MC_BR_ReadParID_0.Busy == TRUE) { }

				/* If mc_br_readparid error */
					if (inst->internal.MC_BR_ReadParID_0.Error == TRUE)
					{
						inst->internal.MC_BR_ReadParID_0.Execute = FALSE;
						inst->internal.AxisReadStep = 0;
					}
				inst->internal.AxisReadStep = 0;
				}
				else {
					inst->internal.AxisReadStep = 0;
					inst->status.ActLagError = 0;
				}
    break;
  }

  MC_BR_BrakeOperation(&inst->internal.MC_BR_BrakeOperation_0);
  MC_BR_ReadParID(&inst->internal.MC_BR_ReadParID_0);
  MC_BR_WriteParID(&inst->internal.MC_BR_WriteParID_0);
		MC_BR_GetHardwareInfo(&inst->internal.MC_BR_GetHardwareInfo_0);
 }
}
```

### Vstupy.var
```iecst
VAR
	diMeranie_PoruchaOtacRotora : BOOL;
	diValcovanie_PoruchaOtacRotora : BOOL;
	diStol_PoruchaOtacStola : BOOL;
	diStol_TeplotaMotoraOK : BOOL;
	diStol_NaliatokOdstrihnuty : BOOL;
	diPoruchaNapajaniaSERVO1 : BOOL;
	diHydraulika_PoruchaCerpadla : BOOL;
	diHydraulika_HladinaOlejaOK : BOOL;
	diHydraulika_TeplotaOlejaOK : BOOL;
	diBZ1_DvereZavrete : BOOL;
	diBZ2_DvereZavrete : BOOL;
	diBZ3_DvereZavrete : BOOL;
	diBZ4_DvereZavrete : BOOL;
	diBZ5_DvereZavrete : BOOL;
	diStavReleKA100_KA101 : BOOL;
	diStavReleKA102_KA103 : BOOL;
	diStavReleKA104_KA105 : BOOL;
	diStav_PrivodVzduchuKanalA : BOOL;
	diStav_PrivodVzduchuKanalB : BOOL;
	diBZ6_DvereZavrete : BOOL;
	diHlavnyPrivodVzduchu_TlakOK : BOOL; (*TLK-1*)
	diHydraulika_Stav_FilterZaneseny : BOOL;
	diTlacitko_RotorOK : BOOL;
	diTlacitko_RotorNG : BOOL;
	diStol_SnimacPolohyStola : BOOL; (*IS-1*)
	diRazenie_ZdvihSpodnaPoloha : BOOL; (*IS-3*)
	diRazenie_PritomnostRotora : BOOL; (*OS-3*)
	diRazenie_ZdvihHornaPoloha : BOOL; (*OS-2*)
	diValcovanie_HornyLimitSnimac : BOOL; (*OS-14*)
	diValcovanie_SpodnyLimitSnimac : BOOL; (*OS-15*)
	diValcovanie_PritomnostRotora : BOOL; (*OS-4*)
	diValcovanie_GriperOtvoreny : BOOL; (*MS-5.1*)
	diValcovanie_GriperZatvoreny : BOOL; (*MS-5.2*)
	diValcovanie_HladinaOlejaOK : BOOL;
	diValcovanie_ZdvihHornaPoloha : BOOL; (*MS-4.2*)
	diValcovanie_ZdvihSpodnaPoloha : BOOL; (*MS-4.1*)
	diValcovanie_PritomnostNastroja : BOOL;
	diValc2_TlakPritlaku_OK : BOOL;
	diValc2_PritomnostRotora : BOOL;
	diValc2_SpomalenieZdvihu : BOOL;
	diValc2_PritlakZasunuty : BOOL;
	diValc2_PritlakVysunuty : BOOL;
	diValc2_ZdvihSpodnyLimit : BOOL;
	diValc2_ZdvihHornyLimit : BOOL;
	diValc2_ZdvihRotoraZasunuty : BOOL;
	diValc2_PorMotoraOtacania : BOOL;
	diValc2_OdbrzdOtacNastrojaRuka : BOOL;
	diValc2_OdbrzdOtacNastrojaMenic : BOOL;
	diValc2_SnimacOtacaniaNastroja : BOOL;
	diValc2_PorNapajaniaServa : BOOL;
	diMeranie_ZdvihSpodnaPoloha : BOOL; (*MS-6*)
	diMeranie_ZdvihHornaPoloha : BOOL; (*OS-5*)
	diMeranie_PritomnostRotora : BOOL; (*OS-6*)
	diMeranie_Osciloskop_Stav_OK : BOOL;
	diMeranie_Osciloskop_Stav_NG : BOOL;
	diStol_PritomnostRotoraVstup : BOOL; (*OS-12*)
	diStol_PritomnostRotoraVystup : BOOL; (*OS-13*)
	diVstupManipul_ZasunutyHore : BOOL; (*MS-7.1*)
	diVstupManipul_VysunutyDole : BOOL; (*MS-7.2*)
	diVstupManipul_PrednyLimitSnimac : BOOL; (*OS-7*)
	diVstupManipul_ZadnyLimitSnimac : BOOL; (*OS-8*)
	diVstupManipul_GriperOtvoreny : BOOL; (*MS-8.1*)
	diVstupManipul_GriperZatvoreny : BOOL; (*MS-8.2*)
	diVstupManipul_ZdvihStredPoloha : BOOL; (*MS-7.3*)
	diVstupManipul_PritomnostNGKusu : BOOL;
	diVstupManipul_SpodSnimacNG_Kusu : BOOL;
	diVstupManipul_HornSnimacNG_Kusu : BOOL;
	diVystupManipul_ZasunutyHore : BOOL; (*MS-9.1*)
	diVystupManipul_ZdvihStredPoloha : BOOL; (*MS-9.3*)
	diVystupManipul_ZadnyLimSnimac : BOOL; (*OS-10*)
	diVystupManipul_PrednyLimSnimac : BOOL; (*OS-9*)
	diVystupManipul_GriperOtvoreny : BOOL; (*MS-10.1*)
	diVystupManipul_GriperZatvoreny : BOOL; (*MS-10.2*)
	diVystupManipul_VysunutyDole : BOOL; (*MS-9.2*)
	diVystDoprOK_SnimacZaplnTrate : BOOL; (*IS-5*)
	diVystDoprNG_SnimacZaplnTrate : BOOL; (*IS-6*)
	diVystDopr_OdsuvacZasunuty : BOOL; (*MS-12.2*)
	diVystDopr_OdsuvacVysunuty : BOOL; (*MS-12.1*)
	diVstupDopr_PritomnostRotora : BOOL; (*IS-4*)
	diOddelovac_PoziciaNavazanie : BOOL; (*MS-11.1*)
	diOddelovac_PoziciaVyvazanie : BOOL; (*MS-11.2*)
	diOddelovac_PritomnostRotora : BOOL; (*OS-11*)
	diVstupDopr_ZdvihRotora_HORE : BOOL;
	diVstupDopr_ZdvihRotora_DOLE : BOOL;
END_VAR
```

### Vystupy.var
```iecst
VAR
	doHydraulika_ChodCerpadla : BOOL;
	doBZ1_ZamkniZamok : BOOL;
	doBZ2_ZamkniZamok : BOOL;
	doBZ3_ZamkniZamok : BOOL;
	doBZ4_ZamkniZamok : BOOL;
	doBZ5_ZamkniZamok : BOOL;
	doBZ6_ZamkniZamok : BOOL;
	doValcovanie_DavkaOleja : BOOL;
	doValc2_DavkaOleja : BOOL;
	doValc2_ZdvihPritlakuHORE : BOOL;
	doValc2_ZostupPritlakuDOLE : BOOL;
	doValc2_BrzdaOtacNastroja : BOOL;
	doMajak_CerveneSvetlo : BOOL;
	doMajak_ZlteSvetlo : BOOL;
	doMajak_ZeleneSvetlo : BOOL;
	doMajak_Hukacka : BOOL;
	doKontrolkaPORUCHA : BOOL;
	doStol_ResetPoruchy : BOOL;
	doZelenaLED_Tlacitko_rotor_OK : BOOL;
	doCervenaLED_Tlacitko_rotor_NG : BOOL;
	doLEDosvetlenie_ZeleneSvetlo : BOOL;
	doLEDosvetlenie_CerveneSvetlo : BOOL;
	doLEDosvetlenie_ModreSvetlo : BOOL;
	doLEDosvetlenie_BieleSvetlo : BOOL;
	doZatvorenieOdvzdHydrauliky : BOOL;
	doStol_OtacajVPRED : BOOL;
	doStol_OtacajVZAD : BOOL;
	doStol_ODBRZDENIE : BOOL;
	doRazenie_ZdvihRotora : BOOL; (*Hydraulika*)
	doRazenie_ZostupRotora : BOOL; (*Hydraulika*)
END_VAR
(***********Ventilový terminál****************************)
VAR
	doOddelovac_PrepniPozNavazania : BOOL; (*YV-1.1*)
	doOddelovac_PrepniPozVyvazania : BOOL; (*YV-1.2*)
	doVstupManipul_ZDVIH : BOOL; (*YV-2.1*)
	doVstupManipul_ZOSTUP : BOOL; (*YV-2.2*)
	doVstupManipul_GriperZATVOR : BOOL; (*YV-3.1*)
	doVstupManipul_GriperOTVOR : BOOL; (*YV-3.2*)
	doVystupManipul_ZDVIH : BOOL; (*YV-4.1*)
	doVystupManipul_ZOSTUP : BOOL; (*YV-4.2*)
	doVystupManipul_GriperZATVOR : BOOL; (*YV-5.1*)
	doVystupManipul_GriperOTVOR : BOOL; (*YV-5.2*)
	doVystDopr_OdsuvacVYSUN : BOOL; (*YV-6.1*)
	doVystDopr_OdsuvacZASUN : BOOL; (*YV-6.2*)
	doValcovanie_ZDVIH_Rotora : BOOL; (*YV-10.1*)
	doValcovanie_ZOSTUP_Rotora : BOOL; (*YV-10.2*)
	doValcovanie_GriperOTVOR : BOOL; (*YV-11.1*)
	doValcovanie_GriperZATVOR : BOOL; (*YV-11.2*)
	doMeranie_ZDVIH : BOOL; (*YV-12.1*)
	doMeranie_ZOSTUP : BOOL; (*YV-12.2*)
	doMeranie_Osciloskop_START : BOOL;
	doMeranie_Osciloskop_STOP : BOOL;
	doMeranie_Osciloskop_Frekvencia : BOOL;
	doVstupDopr_VysunZdvihRotora : BOOL; (*YV-13.1*)
END_VAR
```

### SafetyVstupy.var
```iecst
VAR
	siCS_KanalA : BOOL;
	siCS_KanalB : BOOL;
	siServisneDvere1_KanalA : BOOL;
	siServisneDvere1_KanalB : BOOL;
	siServisneDvere2_KanalA : BOOL;
	siServisneDvere2_KanalB : BOOL;
	siServisneDvere3_KanalA : BOOL;
	siServisneDvere3_KanalB : BOOL;
	siServisneDvere4_KanalA : BOOL;
	siServisneDvere4_KanalB : BOOL;
	siServisneDvere5_KanalA : BOOL;
	siServisneDvere5_KanalB : BOOL;
	siServisneDvere6_KanalA : BOOL;
	siServisneDvere6_KanalB : BOOL;
END_VAR
```

### SafetyVystupy.var
```iecst
VAR
	soMotory : BOOL; (*relé KA100,KA101*)
	soVystupy : BOOL; (*relé KA102,KA103*)
	soKomunikacia_StavCS : BOOL; (*relé KA104,KA105*)
END_VAR
```

### Program Logical/Program/Main (IEC)

#### Main.st - Init, cyclic, exit code
```iecst
PROGRAM _INIT
	Slider:= 0;
	//0 - tlačítko zobrazené, 1 - tlačítko skryté//
	TP_ZobrazPopUpPrihlasenie:= 1;
	TP_ZobrazHlasenieResetZariadenia:= 1;
	TP_ZobrazHlasenieNizkaHladOleja:= 1;
	TP_ZobrazHlasenieZamkyVyblokov:= 1;
	VnutorneValcovanie_AKTIVNE:= TRUE;
	VonkajsieValcovanie_AKTIVNE:= FALSE;

END_PROGRAM

PROGRAM _CYCLIC

	//Volanie podprogramov//
	ZobrazenieTlacitok;
	OvladanieHydrauliky;
	OvladanieSafety;

	//Ovládanie osvetlenia bunky//
	IF NOT diBZ1_DvereZavrete OR NOT diBZ2_DvereZavrete OR NOT diBZ3_DvereZavrete OR NOT diBZ4_DvereZavrete OR NOT diBZ5_DvereZavrete OR NOT diBZ6_DvereZavrete THEN
		doLEDosvetlenie_BieleSvetlo:= TRUE;
		doLEDosvetlenie_ZeleneSvetlo:= FALSE;
		doLEDosvetlenie_CerveneSvetlo:= FALSE;
	ELSIF NastalaPorucha THEN
		doLEDosvetlenie_CerveneSvetlo:= TRUE;
		doLEDosvetlenie_BieleSvetlo:= FALSE;
		doLEDosvetlenie_ZeleneSvetlo:= FALSE;
	ELSIF Zariadenie_StavAutomat THEN
		doLEDosvetlenie_ZeleneSvetlo:= TRUE;
		doLEDosvetlenie_BieleSvetlo:= FALSE;
		doLEDosvetlenie_CerveneSvetlo:= FALSE;
	ELSE
		doLEDosvetlenie_BieleSvetlo:= FALSE;
		doLEDosvetlenie_ZeleneSvetlo:= FALSE;
		doLEDosvetlenie_CerveneSvetlo:= FALSE;
	END_IF

	//Zobrazenie úvodnej obrazovky//
	IF NOT SafetyPLC_Nabehlo THEN
		CisloZadanejObrazovky:= 0;
		IF EDGEPOS (Blikac500ms = TRUE) THEN
			Slider:= Slider+1;
			IF Slider > 10 THEN
				Slider:= 0;
			END_IF
		END_IF
	END_IF

	//Prepnutie na hlavnú obrazovku//
	IF EDGEPOS (SafetyPLC_Nabehlo = TRUE) THEN
		CisloZadanejObrazovky:= 1;
	ELSIF EDGENEG(BezpOkruhOplotenia_Aktivovany = TRUE) AND CisloAktualnejObrazovky <> 100 THEN
		CisloZadanejObrazovky:= 1;
	ELSIF SafetyPLC_Nabehlo AND CisloAktualnejObrazovky = 0 THEN
		CisloZadanejObrazovky:= 1;
	END_IF

	//Prepnutie na hlavnú obrazovku ručného režimu pri poruche//
//	IF EDGEPOS (NastalaPorucha = TRUE) THEN
//		IF Zariadenie_StavManual AND CisloAktualnejObrazovky <> 20 THEN
//			CisloZadanejObrazovky:= 20;
//		END_IF
//	END_IF

	//Prepnutie na obrazovku alarmov pri poruche//
	IF EDGEPOS (NastalaPorucha) THEN
		CisloZadanejObrazovky:= 102;
	END_IF

	//Zariadenie stav Homing OK//
	IF VstupManipulator_HomingOK AND Valcovanie_HomingOK AND VystupManipulator_HomingOK AND Valcovanie2_HomingOK THEN
		Zariadenie_HomingOK:= TRUE;
	ELSE
		Zariadenie_HomingOK:= FALSE;
	END_IF

	//Zariadenie stav Automat//
	IF Meranie_Automat OR Oddelovac_Automat OR ZdvihRotora_Automat OR Razenie_Automat OR Stol_Automat OR Strihanie_Automat OR Valcovanie_Automat OR Valcovanie2_Automat OR VstupManipulator_Automat OR VystupManipulator_Automat OR VystupOdsuvac_Automat THEN
		Zariadenie_StavAutomat:= TRUE;
	ELSE
		Zariadenie_StavAutomat:= FALSE;
		Zariadenie_PrebiehaUkoncenie:= FALSE;
		Zariadenie_PrebiehaKoniecCyklu:= FALSE;
		Zariadenie_PrebiehaRevorkRezim:= FALSE;
	END_IF

	//Zariadenie stav Manual//
	IF Meranie_Manual OR Oddelovac_Manual OR ZdvihRotora_Manual OR Razenie_Manual OR Stol_Manual OR Strihanie_Manual OR Valcovanie_Manual OR Valcovanie2_Manual OR VstupManipulator_Manual OR VystupManipulator_Manual OR VystupOdsuvac_Manual THEN
		Zariadenie_StavManual:= TRUE;
	ELSE
		Zariadenie_StavManual:= FALSE;
	END_IF

	//Zariadenie stav po inicializacii//
	IF Meranie_PoINIT AND Oddelovac_PoINIT AND ZdvihRotora_PoINIT AND Razenie_PoINIT AND Stol_PoINIT AND Strihanie_PoINIT AND Valcovanie_PoINIT AND Valcovanie2_PoINIT AND VstupManipulator_PoINIT AND VystupManipulator_PoINIT AND VystupOdsuvac_PoINIT THEN
		Zariadenie_StavPoINIT:= TRUE;
	ELSE
		Zariadenie_StavPoINIT:= FALSE;
	END_IF

	//Zariadenie stav prebieha homing//
	IF VstupManipulator_PrebiehaHoming OR Valcovanie_PrebiehaHoming OR Valcovanie2_PrebiehaHoming OR VystupManipulator_PrebiehaHoming THEN
		Zariadenie_PrebiehaHoming:= TRUE;
	ELSE
		Zariadenie_PrebiehaHoming:= FALSE;
	END_IF

	//Zariadenie stav moduly OK//
	IF Modul_DB1_OK AND Modul_DB2_OK AND Modul_DB3_OK AND Modul_DB4_OK AND Modul_DB5_OK AND Modul_DB6_OK THEN
		Zariadenie_Moduly_OK:= TRUE;
	ELSE
		Zariadenie_Moduly_OK:= FALSE;
	END_IF

	//Spustenie výroby na zariadení//
	IF Zariadenie_Automat AND BezpOkruhOplotenia_Aktivovany THEN
		Meranie_Automat:= TRUE;
		Oddelovac_Automat:= TRUE;
		ZdvihRotora_Automat:= TRUE;
		Razenie_Automat:= TRUE;
		Stol_Automat:= TRUE;
		Strihanie_Automat:= TRUE;
		Valcovanie_Automat:= TRUE;
		Valcovanie2_Automat:= TRUE;
		VstupManipulator_Automat:= TRUE;
		VystupManipulator_Automat:= TRUE;
		VystupOdsuvac_Automat:= TRUE;
		Zariadenie_Automat:= FALSE;
	ELSIF Zariadenie_Automat AND NOT BezpOkruhOplotenia_Aktivovany THEN
		Zariadenie_Automat:= FALSE;
	END_IF

	//Spustenie revork režimu//
	IF Zariadenie_RevorkRezim AND BezpOkruhOplotenia_Aktivovany THEN
		Meranie_Automat:= TRUE;
		Oddelovac_Automat:= TRUE;
		ZdvihRotora_Automat:= TRUE;
		Razenie_Automat:= TRUE;
		Stol_Automat:= TRUE;
		Strihanie_Automat:= TRUE;
		Valcovanie_Automat:= TRUE;
		Valcovanie2_Automat:= TRUE;
		VstupManipulator_Automat:= TRUE;
		VystupManipulator_Automat:= TRUE;
		VystupOdsuvac_Automat:= TRUE;
		Zariadenie_PrebiehaRevorkRezim:= TRUE;
		Zariadenie_RevorkRezim:= FALSE;
	ELSIF Zariadenie_RevorkRezim AND NOT BezpOkruhOplotenia_Aktivovany THEN
		Zariadenie_RevorkRezim:= FALSE;
	END_IF

	//Vypnutie ručného režimu na hlavnej obrazovke ručného režimu//
	IF EDGEPOS(CisloAktualnejObrazovky = 20) THEN
		Meranie_Manual:= FALSE;
		Oddelovac_Manual:= FALSE;
		ZdvihRotora_Manual:= FALSE;
		Razenie_Manual:= FALSE;
		Stol_Manual:= FALSE;
		Strihanie_Manual:= FALSE;
		Valcovanie_Manual:= FALSE;
		Valcovanie2_Manual:= FALSE;
		VstupManipulator_Manual:= FALSE;
		VystupManipulator_Manual:= FALSE;
		VystupOdsuvac_Manual:= FALSE;
	END_IF

	//Ukončenie výroby na zariadení//
	IF Zariadenie_KoniecVyroby THEN
		Meranie_KoniecVyroby:= TRUE;
		Oddelovac_KoniecVyroby:= TRUE;
		ZdvihRotora_KoniecVyroby:= TRUE;
		Razenie_KoniecVyroby:= TRUE;
		Stol_KoniecVyroby:= TRUE;
		Strihanie_KoniecVyroby:= TRUE;
		Valcovanie_KoniecVyroby:= TRUE;
		Valcovanie2_KoniecVyroby:= TRUE;
		VstupManipulator_KoniecVyroby:= TRUE;
		VystupManipulator_KoniecVyroby:= TRUE;
		VystupOdsuvac_KoniecVyroby:= TRUE;
		Zariadenie_PrebiehaUkoncenie:= TRUE;
		Zariadenie_KoniecVyroby:= FALSE;
	END_IF

	//Ukončenie pracovného cyklu//
	IF EDGEPOS(NastalaPorucha = TRUE) THEN
		Zariadenie_KoniecCyklu:= TRUE;
	END_IF

	IF Zariadenie_KoniecCyklu THEN
		Oddelovac_KoniecCyklu:= TRUE;
		ZdvihRotora_KoniecCyklu:= TRUE;
		VstupManipulator_KoniecCyklu:= TRUE;
		Strihanie_KoniecCyklu:= TRUE;
		Razenie_KoniecCyklu:= TRUE;
		Valcovanie_KoniecCyklu:= TRUE;
		Valcovanie2_KoniecCyklu:= TRUE;
		Meranie_KoniecCyklu:= TRUE;
		Stol_KoniecCyklu:= TRUE;
		VystupManipulator_KoniecCyklu:= TRUE;
		VystupOdsuvac_KoniecCyklu:= TRUE;
		Zariadenie_PrebiehaKoniecCyklu:= TRUE;
		Zariadenie_KoniecCyklu:= FALSE;
	END_IF

	//Resetovanie zariadenia//
	IF Zariadenie_Reset THEN
		Meranie_Reset:= TRUE;
		Oddelovac_Reset:= TRUE;
		ZdvihRotora_Reset:= TRUE;
		Razenie_Reset:= TRUE;
		Stol_Reset:= TRUE;
		Strihanie_Reset:= TRUE;
		Valcovanie_Reset:= TRUE;
		Valcovanie2_Reset:= TRUE;
		VstupManipulator_Reset:= TRUE;
		VystupManipulator_Reset:= TRUE;
		VystupOdsuvac_Reset:= TRUE;
		Zariadenie_Reset:= FALSE;
	END_IF

END_PROGRAM

PROGRAM _EXIT
			(* Insert code here *)

			END_PROGRAM
```

#### Variables.var - Local variables
```iecst
VAR
	CasZaplneniaDopravnikaNG : TON;
	CasZaplneniaDopravnikaOK : TON;
	CasPredResetomOplotenia : TON;
	CasNizkaHladinaOleja : TON;
	CasZapnutiaHydrauliky : TON;
END_VAR
```

#### ZobrazenieTlacitok.st
```iecst
ACTION ZobrazenieTlacitok:

	//Zamknutie tlačítka Manuálny režimm//
	IF BezpOkruhOplotenia_Aktivovany AND NOT NastalaPorucha AND Stav_ServaREADY AND Zariadenie_Moduly_OK THEN
		TP_ZamkniTlacitkoRezimManual:= 0;
	ELSE
		TP_ZamkniTlacitkoRezimManual:= 1;
	END_IF

	//Zamknutie tlačítka Automatický režim//
	IF BezpOkruhOplotenia_Aktivovany AND NOT NastalaPorucha AND Stav_ServaREADY AND Zariadenie_Moduly_OK THEN
		TP_ZamkniTlacitkoRezimAutomat:= 0;
	ELSE
		TP_ZamkniTlacitkoRezimAutomat:= 1;
	END_IF

	//Zamknutie tlačítka Revork režim//
	IF NOT BezpOkruhOplotenia_Aktivovany THEN
		TP_ZamkniTlacitkoRezimRevork:= 1;
	ELSIF NastalaPorucha THEN
		TP_ZamkniTlacitkoRezimRevork:= 1;
	ELSIF NOT VnutorneValcovanie_AKTIVNE AND NOT VonkajsieValcovanie_AKTIVNE THEN
		TP_ZamkniTlacitkoRezimRevork:= 1;
	ELSIF Zariadenie_StavAutomat THEN
		TP_ZamkniTlacitkoRezimRevork:= 1;
	ELSE
		TP_ZamkniTlacitkoRezimRevork:= 0;
	END_IF

	//Zamknutie tlačítok aktivácie valcovania//
	IF Zariadenie_StavAutomat THEN
		TP_ZamkniTlacitkaAktivValcovania:= 1;
	ELSE
		TP_ZamkniTlacitkaAktivValcovania:= 0;
	END_IF

	//Zamknutie tlačítka Štart Automat//
	IF BezpOkruhOplotenia_Aktivovany AND NOT NastalaPorucha AND NOT Zariadenie_StavPoINIT AND NOT Zariadenie_PrebiehaUkoncenie AND Stav_ServaREADY AND Zariadenie_Moduly_OK AND VnutorneValcovanie_AKTIVNE AND NOT Zariadenie_PrebiehaRevorkRezim THEN
		TP_ZamkniTlacStartAutomat:= 0;
	ELSE
		TP_ZamkniTlacStartAutomat:= 1;
	END_IF

	//Blikanie tlačítka Štart Automat//
	IF Zariadenie_StavAutomat AND NOT Zariadenie_StavPoINIT THEN
		BlikanieTlacitkaStartZariadenia:= Blikac500ms;
	ELSIF Zariadenie_StavAutomat AND Zariadenie_StavPoINIT THEN
		BlikanieTlacitkaStartZariadenia:= 1;
	ELSE
		BlikanieTlacitkaStartZariadenia:= 0;
	END_IF

	//Zamknutie tlačítka Ukončenie výroby//
	IF Zariadenie_StavPoINIT AND NOT Zariadenie_PrebiehaUkoncenie AND NOT Zariadenie_PrebiehaKoniecCyklu THEN
		TP_ZamkniTlacUkoncenieVyroby:= 0;
	ELSE
		TP_ZamkniTlacUkoncenieVyroby:= 1;
	END_IF

	//Zamknutie tlačítka Koniec cyklu//
	IF Zariadenie_StavPoINIT AND NOT Zariadenie_PrebiehaKoniecCyklu THEN
		TP_ZamkniTlacKoniecCyklu:= 0;
	ELSE
		TP_ZamkniTlacKoniecCyklu:= 1;
	END_IF

	//Zobrazenie tlačítka Home//
	IF Zariadenie_StavAutomat THEN
		TP_ZobrazTlacitkoHome:= 1;
	ELSIF FM_Menic[3].Output.Status.Running THEN
		TP_ZobrazTlacitkoHome:= 1;
	ELSE
		TP_ZobrazTlacitkoHome:= 0;
	END_IF

	//Zobrazenie hlásenia NG dopravník plný//
	IF diVystDoprNG_SnimacZaplnTrate THEN
		CasZaplneniaDopravnikaNG.IN:= TRUE;
	ELSE
		CasZaplneniaDopravnikaNG.IN:= FALSE;
	END_IF

	IF CasZaplneniaDopravnikaNG.Q THEN
		TP_ZobrazHlasenieDoprNG_Plny:= 0;
	ELSE
		TP_ZobrazHlasenieDoprNG_Plny:= 1;
	END_IF

	CasZaplneniaDopravnikaNG.PT:= T#5s;
	CasZaplneniaDopravnikaNG();

	//Zobrazenie hlásenia OK dopravník plný//
	IF diVystDoprOK_SnimacZaplnTrate THEN
		CasZaplneniaDopravnikaOK.IN:= TRUE;
	ELSE
		CasZaplneniaDopravnikaOK.IN:= FALSE;
	END_IF

	IF CasZaplneniaDopravnikaOK.Q THEN
		TP_ZobrazHlasenieDoprOK_Plny:= 0;
	ELSE
		TP_ZobrazHlasenieDoprOK_Plny:= 1;
	END_IF

	CasZaplneniaDopravnikaOK.PT:= T#5s;
	CasZaplneniaDopravnikaOK();

	//Zobrazenie hlásenia nízka hladina oleja//
	IF NOT diValcovanie_HladinaOlejaOK THEN
		CasNizkaHladinaOleja.IN:= TRUE;
	ELSE
		CasNizkaHladinaOleja.IN:= FALSE;
	END_IF

	IF CasNizkaHladinaOleja.Q THEN
		TP_ZobrazHlasenieNizkaHladOleja:= 0;
	ELSE
		TP_ZobrazHlasenieNizkaHladOleja:= 1;
	END_IF

	CasNizkaHladinaOleja.PT:= T#5s;
	CasNizkaHladinaOleja();

	//Zobrazenie hlásenia - zámky vyblokované//
	IF RezimServis THEN
		TP_ZobrazHlasenieZamkyVyblokov:= 0;
	ELSE
		TP_ZobrazHlasenieZamkyVyblokov:= 1;
	END_IF

	//Vstupný manipulátor - zamknutie pojazdu //
	IF VstupManipulator_HomingOK AND diVstupManipul_ZasunutyHore THEN
		TP_VstupManip_ZamkniTlacPojazdu:= 0;
	ELSE
		TP_VstupManip_ZamkniTlacPojazdu:= 1;
	END_IF

	//Stanica strihania - zamknutie zdvihu rotora//
	IF diStol_SnimacPolohyStola AND Vyrazanie.IN.UchytenieNaliatkuOtvorene AND NOT Vyrazanie.IN.UchytenieNaliatkuZatvorene AND Vyrazanie.IN.OdhadzovanieJeVpredu AND Vyrazanie.IN.OdhadzovanieJeVpredu2 AND Vyrazanie.IN.UchytenieKolikaOtvorene AND NOT Vyrazanie.IN.UchytenieKolikaZatvorene THEN
		TP_Strihanie_ZamkniZdvihRotora:= 0;
	ELSE
		TP_Strihanie_ZamkniZdvihRotora:= 1;
	END_IF

	//Stanica razenia - zamknutie zdvihu rotora//
	IF diStol_SnimacPolohyStola THEN
		TP_Razenie_ZamkniZdvihRotora:= 0;
	ELSE
		TP_Razenie_ZamkniZdvihRotora:= 1;
	END_IF

	//Stanica valcovania - zamknutie zdvihu rotora//
	IF diStol_SnimacPolohyStola AND diValcovanie_GriperOtvoreny THEN
		TP_Valcovanie_ZamkniZdvihRotora:= 0;
	ELSE
		TP_Valcovanie_ZamkniZdvihRotora:= 1;
	END_IF

	//Stanica valcovania - zamknutie zdvihu nástroja//
	IF Valcovanie_HomingOK THEN
		TP_Valcovanie_ZamkniZdvihServa:= 0;
	ELSE
		TP_Valcovanie_ZamkniZdvihServa:= 1;
	END_IF

	//Stanica valcovania 2 - zamknutie zdvihu rotora//
	IF NOT Valcovanie2_HomingOK THEN
		TP_Valcovanie2_ZamkniZdvihServa:= 1;
	ELSIF Valcovanie2_AktualPozMM >= Valcovanie2_ZadanaPozMM THEN
		TP_Valcovanie2_ZamkniZdvihServa:= 1;
	ELSE
		TP_Valcovanie2_ZamkniZdvihServa:= 0;
	END_IF

	//Stanica valcovania 2 - zamknutie zostupu rotora//
	IF NOT Valcovanie2_HomingOK THEN
		TP_Valcovanie2_ZamkniZostupServa:= 1;
	ELSIF Valcovanie2_AktualPozMM <= 13 THEN
		TP_Valcovanie2_ZamkniZostupServa:= 1;
	ELSE
		TP_Valcovanie2_ZamkniZostupServa:= 0;
	END_IF

	//Stol - zamknutie otáčania//
	IF NOT Stol_BlokovanieOtacania THEN
		TP_Stol_ZamkniOtacanie:= 0;
	ELSE
		TP_Stol_ZamkniOtacanie:= 1;
	END_IF

	//Stanica merania - zamknutie zdvihu rotora//
	IF diStol_SnimacPolohyStola THEN
		TP_Meranie_ZamkniZdvihRotora:= 0;
	ELSE
		TP_Meranie_ZamkniZdvihRotora:= 1;
	END_IF

	//Výstupný manipulátor - zamknutie pojazdu//
	IF VystupManipulator_HomingOK AND diVystupManipul_ZasunutyHore THEN
		TP_VystupManip_ZamkniTlacPojazdu:= 0;
	ELSE
		TP_VystupManip_ZamkniTlacPojazdu:= 1;
	END_IF

	//Výstupný odsúvač - zamknutie vysunutia//
	IF diVystupManipul_ZasunutyHore THEN
		TP_VystOdsuvac_ZamkniTlacVysunut:= 0;
	ELSE
		TP_VystOdsuvac_ZamkniTlacVysunut:= 1;
	END_IF

	//Zamknutie zámkov oplotenia//
	IF Zariadenie_StavAutomat THEN
		TP_ZamkniTlacitkaZamkovOplotenia:= 1;
	ELSIF FM_Menic[3].Output.Status.Running THEN
		TP_ZamkniTlacitkaZamkovOplotenia:= 1;
	ELSE
		TP_ZamkniTlacitkaZamkovOplotenia:= 0;
	END_IF

	//Zamknutie tlačítka servis//
	IF ZvolenaUroven = 1000 THEN
		TP_ZamkniTlacitkoServis:= 0;
	ELSE
		TP_ZamkniTlacitkoServis:= 1;
		RezimServis:= FALSE;
	END_IF

	//***************************************Zamknutie parametrov nastavenia zariadenia***************************************************************//
	IF ZvolenaUroven < 10 THEN
		TP_ZamkniParametreUrovenOperator:= 2;
	ELSE
		TP_ZamkniParametreUrovenOperator:= 0;
	END_IF

	IF ZvolenaUroven < 20 THEN
		TP_ZamkniParametreUrovenServisak:= 2;
	ELSE
		TP_ZamkniParametreUrovenServisak:= 0;
	END_IF

	//0-sivá, 1- žltá, 2- zelená, 3- červená//
	//Stav vstupného oddelovača//
	IF PoruchaOddelovaca THEN
		StavOddelovaca:= 3;
	ELSIF NOT Oddelovac_Automat THEN
		StavOddelovaca:= 0;
	ELSIF Oddelovac_Automat AND NOT Oddelovac_PoINIT THEN
		StavOddelovaca:= 1;
	ELSIF Oddelovac_Automat AND Oddelovac_PoINIT THEN
		StavOddelovaca:= 2;
	END_IF

	//Stav zdvihu rotora na vstupnom dopravníku//
	IF PoruchaZdvihuRotora THEN
		StavZdvihuRotora:= 3;
	ELSIF NOT ZdvihRotora_Automat THEN
		StavZdvihuRotora:= 0;
	ELSIF ZdvihRotora_Automat AND NOT ZdvihRotora_PoINIT THEN
		StavZdvihuRotora:= 1;
	ELSIF ZdvihRotora_Automat AND ZdvihRotora_PoINIT THEN
		StavZdvihuRotora:= 2;
	END_IF

	//Stav vstupného manipulátora//
	IF PoruchaVstupManipulator THEN
		StavVstupnehoManipulatora:= 3;
	ELSIF NOT VstupManipulator_Automat THEN
		StavVstupnehoManipulatora:= 0;
	ELSIF VstupManipulator_Automat AND NOT VstupManipulator_PoINIT THEN
		StavVstupnehoManipulatora:= 1;
	ELSIF VstupManipulator_Automat AND VstupManipulator_PoINIT THEN
		StavVstupnehoManipulatora:= 2;
	END_IF

	//Stav stola//
	IF PoruchaOtocnyStol THEN
		StavStola:= 3;
	ELSIF NOT Stol_Automat THEN
		StavStola:= 0;
	ELSIF Stol_Automat AND NOT Stol_PoINIT THEN
		StavStola:= 1;
	ELSIF Stol_Automat AND Stol_PoINIT THEN
		StavStola:= 2;
	END_IF

	//Stav strihania//
	IF PoruchaStanicaStrihania THEN
		StavStrihania:= 3;
	ELSIF NOT Strihanie_Automat THEN
		StavStrihania:= 0;
	ELSIF Strihanie_Automat AND NOT Strihanie_PoINIT THEN
		StavStrihania:= 1;
	ELSIF Strihanie_Automat AND Strihanie_PoINIT THEN
		StavStrihania:= 2;
	END_IF

	//Stav razenia//
	IF PoruchaStanicaRazenia THEN
		StavRazenia:= 3;
	ELSIF NOT Razenie_Automat THEN
		StavRazenia:= 0;
	ELSIF Razenie_Automat AND NOT Razenie_PoINIT THEN
		StavRazenia:= 1;
	ELSIF Razenie_Automat AND Razenie_PoINIT THEN
		StavRazenia:= 2;
	END_IF

	//Stav valcovania//
	IF PoruchaStanicaValcovania THEN
		StavValcovania:= 3;
	ELSIF NOT Valcovanie_Automat THEN
		StavValcovania:= 0;
	ELSIF Valcovanie_Automat AND NOT Valcovanie_PoINIT THEN
		StavValcovania:= 1;
	ELSIF Valcovanie_Automat AND Valcovanie_PoINIT THEN
		StavValcovania:= 2;
	END_IF

	//Stav valcovania 2//
	IF PoruchaStanicaValcovania2 THEN
		StavValcovania2:= 3;
	ELSIF NOT Valcovanie2_Automat THEN
		StavValcovania2:= 0;
	ELSIF Valcovanie2_Automat AND NOT Valcovanie2_PoINIT THEN
		StavValcovania2:= 1;
	ELSIF Valcovanie2_Automat AND Valcovanie2_PoINIT THEN
		StavValcovania2:= 2;
	END_IF

	//Stav merania//
	IF PoruchaStanicaMerania THEN
		StavMerania:= 3;
	ELSIF NOT Meranie_Automat THEN
		StavMerania:= 0;
	ELSIF Meranie_Automat AND NOT Meranie_PoINIT THEN
		StavMerania:= 1;
	ELSIF Meranie_Automat AND Meranie_PoINIT THEN
		StavMerania:= 2;
	END_IF

	//Stav výstupného manipulátora//
	IF PoruchaVystupManipulator THEN
		StavVystupnehoManipulatora:= 3;
	ELSIF NOT VystupManipulator_Automat THEN
		StavVystupnehoManipulatora:= 0;
	ELSIF VystupManipulator_Automat AND NOT VystupManipulator_PoINIT THEN
		StavVystupnehoManipulatora:= 1;
	ELSIF VystupManipulator_Automat AND VystupManipulator_PoINIT THEN
		StavVystupnehoManipulatora:= 2;
	END_IF

	//Stav výstupného odsúvača//
	IF PoruchaVystupOdsuvac THEN
		StavVystupnehoOdsuvaca:= 3;
	ELSIF NOT VystupOdsuvac_Automat THEN
		StavVystupnehoOdsuvaca:= 0;
	ELSIF VystupOdsuvac_Automat AND NOT VystupOdsuvac_PoINIT THEN
		StavVystupnehoOdsuvaca:= 1;
	ELSIF VystupOdsuvac_Automat AND VystupOdsuvac_PoINIT THEN
		StavVystupnehoOdsuvaca:= 2;
	END_IF

	//Stav bezpečnostného zámku BZ1//
	IF diBZ1_DvereZavrete AND NOT Stav_BZ1_Zamknuty THEN
		StavZamkuBZ1:= Blikac500ms;
	ELSIF diBZ1_DvereZavrete AND Stav_BZ1_Zamknuty THEN
		StavZamkuBZ1:= 2;
	ELSE
		StavZamkuBZ1:= 3;
	END_IF

	//Stav bezpečnostného zámku BZ2//
	IF diBZ2_DvereZavrete AND NOT Stav_BZ2_Zamknuty THEN
		StavZamkuBZ2:= Blikac500ms;
	ELSIF diBZ2_DvereZavrete AND Stav_BZ2_Zamknuty THEN
		StavZamkuBZ2:= 2;
	ELSE
		StavZamkuBZ2:= 3;
	END_IF

	//Stav bezpečnostného zámku BZ3//
	IF diBZ3_DvereZavrete AND NOT Stav_BZ3_Zamknuty THEN
		StavZamkuBZ3:= Blikac500ms;
	ELSIF diBZ3_DvereZavrete AND Stav_BZ3_Zamknuty THEN
		StavZamkuBZ3:= 2;
	ELSE
		StavZamkuBZ3:= 3;
	END_IF

	//Stav bezpečnostného zámku BZ4//
	IF diBZ4_DvereZavrete AND NOT Stav_BZ4_Zamknuty THEN
		StavZamkuBZ4:= Blikac500ms;
	ELSIF diBZ4_DvereZavrete AND Stav_BZ4_Zamknuty THEN
		StavZamkuBZ4:= 2;
	ELSE
		StavZamkuBZ4:= 3;
	END_IF

	//Stav bezpečnostného zámku BZ5//
	IF diBZ5_DvereZavrete AND NOT Stav_BZ5_Zamknuty THEN
		StavZamkuBZ5:= Blikac500ms;
	ELSIF diBZ5_DvereZavrete AND Stav_BZ5_Zamknuty THEN
		StavZamkuBZ5:= 2;
	ELSE
		StavZamkuBZ5:= 3;
	END_IF

	//Stav bezpečnostného zámku BZ6//
	IF diBZ6_DvereZavrete AND NOT Stav_BZ6_Zamknuty THEN
		StavZamkuBZ6:= Blikac500ms;
	ELSIF diBZ6_DvereZavrete AND Stav_BZ6_Zamknuty THEN
		StavZamkuBZ6:= 2;
	ELSE
		StavZamkuBZ6:= 3;
	END_IF

		END_ACTION
```

#### OvladanieSafety.st
```iecst
ACTION OvladanieSafety:

	diStavReleKA100_KA101;
	diStavReleKA102_KA103;
	diStavReleKA104_KA105;
	diStav_PrivodVzduchuKanalA;
	diStav_PrivodVzduchuKanalB;
	Reset_CS;
	Reset_Oplotenia;
	SafetyPLC_Nabehlo;
	BezpOkruhCS_Aktivovany;
	BezpOkruhOplotenia_Aktivovany;
	Stav_CS_Odblokovane;
	Stav_BZ1_Zamknuty;
	Stav_BZ2_Zamknuty;
	Stav_BZ3_Zamknuty;
	Stav_BZ4_Zamknuty;
	Stav_BZ5_Zamknuty;
	Stav_BZ6_Zamknuty;
	RezimServis;

	//Ovladanie dverí č.1//
	IF EDGEPOS (Zamkni_BZ1 = TRUE) AND BezpOkruhCS_Aktivovany THEN
		IF diBZ1_DvereZavrete AND NOT Stav_BZ1_Zamknuty THEN
			doBZ1_ZamkniZamok:= TRUE;
		ELSIF diBZ1_DvereZavrete AND Stav_BZ1_Zamknuty AND NOT Zariadenie_StavAutomat THEN
			doBZ1_ZamkniZamok:= FALSE;
		END_IF
	ELSIF NOT BezpOkruhCS_Aktivovany THEN
		doBZ1_ZamkniZamok:= FALSE;
	END_IF

	//Ovladanie dverí č.2//
	IF EDGEPOS (Zamkni_BZ2 = TRUE) AND BezpOkruhCS_Aktivovany THEN
		IF diBZ2_DvereZavrete AND NOT Stav_BZ2_Zamknuty THEN
			doBZ2_ZamkniZamok:= TRUE;
		ELSIF diBZ2_DvereZavrete AND Stav_BZ2_Zamknuty AND NOT Zariadenie_StavAutomat THEN
			doBZ2_ZamkniZamok:= FALSE;
		END_IF
	ELSIF NOT BezpOkruhCS_Aktivovany THEN
		doBZ2_ZamkniZamok:= FALSE;
	END_IF

	//Ovladanie dverí č.3//
	IF EDGEPOS (Zamkni_BZ3 = TRUE) AND BezpOkruhCS_Aktivovany THEN
		IF diBZ3_DvereZavrete AND NOT Stav_BZ3_Zamknuty THEN
			doBZ3_ZamkniZamok:= TRUE;
		ELSIF diBZ3_DvereZavrete AND Stav_BZ3_Zamknuty AND NOT Zariadenie_StavAutomat THEN
			doBZ3_ZamkniZamok:= FALSE;
		END_IF
	ELSIF NOT BezpOkruhCS_Aktivovany THEN
		doBZ3_ZamkniZamok:= FALSE;
	END_IF

	//Ovladanie dverí č.4//
	IF EDGEPOS (Zamkni_BZ4 = TRUE) AND BezpOkruhCS_Aktivovany THEN
		IF diBZ4_DvereZavrete AND NOT Stav_BZ4_Zamknuty THEN
			doBZ4_ZamkniZamok:= TRUE;
		ELSIF diBZ4_DvereZavrete AND Stav_BZ4_Zamknuty AND NOT Zariadenie_StavAutomat THEN
			doBZ4_ZamkniZamok:= FALSE;
		END_IF
	ELSIF NOT BezpOkruhCS_Aktivovany THEN
		doBZ4_ZamkniZamok:= FALSE;
	END_IF

	//Ovladanie dverí č.5//
	IF EDGEPOS (Zamkni_BZ5 = TRUE) AND BezpOkruhCS_Aktivovany THEN
		IF diBZ5_DvereZavrete AND NOT Stav_BZ5_Zamknuty THEN
			doBZ5_ZamkniZamok:= TRUE;
		ELSIF diBZ5_DvereZavrete AND Stav_BZ5_Zamknuty AND NOT Zariadenie_StavAutomat THEN
			doBZ5_ZamkniZamok:= FALSE;
		END_IF
	ELSIF NOT BezpOkruhCS_Aktivovany THEN
		doBZ5_ZamkniZamok:= FALSE;
	END_IF

	//Ovladanie dverí č.6//
	IF EDGEPOS (Zamkni_BZ6 = TRUE) AND BezpOkruhCS_Aktivovany THEN
		IF diBZ6_DvereZavrete AND NOT Stav_BZ6_Zamknuty THEN
			doBZ6_ZamkniZamok:= TRUE;
		ELSIF diBZ6_DvereZavrete AND Stav_BZ6_Zamknuty AND NOT Zariadenie_StavAutomat THEN
			doBZ6_ZamkniZamok:= FALSE;
		END_IF
	ELSIF NOT BezpOkruhCS_Aktivovany THEN
		doBZ6_ZamkniZamok:= FALSE;
	END_IF

	//Resetovanie oplotenia//
	IF ((Stav_BZ1_Zamknuty AND Stav_BZ2_Zamknuty AND Stav_BZ3_Zamknuty AND Stav_BZ4_Zamknuty AND Stav_BZ5_Zamknuty AND Stav_BZ6_Zamknuty) OR RezimServis) AND BezpOkruhCS_Aktivovany THEN
		CasPredResetomOplotenia.IN:= TRUE;
	ELSE
		CasPredResetomOplotenia.IN:= FALSE;
	END_IF

	IF CasPredResetomOplotenia.Q AND NOT BezpOkruhOplotenia_Aktivovany AND BezpOkruhCS_Aktivovany THEN
		Reset_Oplotenia:= TRUE;
	ELSE
		Reset_Oplotenia:= FALSE;
	END_IF

	CasPredResetomOplotenia.PT:= T#500ms;
	CasPredResetomOplotenia();

	//Podsvietenie tlačítka reset CS//
	IF Stav_CS_Odblokovane AND NOT BezpOkruhCS_Aktivovany THEN
		TP_ModraLEDResetCS:= Blikac500ms;
	ELSIF BezpOkruhCS_Aktivovany THEN
		TP_ModraLEDResetCS:= 2;
	ELSE
		TP_ModraLEDResetCS:= 3;
	END_IF

	//Podsvietenie tlačítka reset oplotenia//
	IF BezpOkruhCS_Aktivovany AND Stav_BZ1_Zamknuty AND Stav_BZ2_Zamknuty AND Stav_BZ3_Zamknuty AND Stav_BZ4_Zamknuty AND Stav_BZ5_Zamknuty AND Stav_BZ6_Zamknuty AND NOT BezpOkruhOplotenia_Aktivovany THEN
		TP_ModraLEDResetOplotenia:= Blikac500ms;
	ELSIF (RezimServis OR BezpOkruhOplotenia_Aktivovany) AND BezpOkruhCS_Aktivovany THEN
		TP_ModraLEDResetOplotenia:= 2;
	ELSE
		TP_ModraLEDResetOplotenia:= 3;
	END_IF

END_ACTION
```

#### OvladanieHydrauliky.st
```iecst
ACTION OvladanieHydrauliky:

	//Ovládanie čerpadla//
	//Zapnutie čerpadla hydrauliky//
	IF (Strihanie_Automat OR Razenie_Automat) AND NOT Stol_StavPrazdnyStol THEN
		CasVypnutiaHydrauliky.IN:= FALSE;
		doZatvorenieOdvzdHydrauliky:= FALSE;
		CasZapnutiaHydrauliky.IN:= TRUE;
	ELSIF Strihanie_Manual OR Razenie_Manual THEN
		CasVypnutiaHydrauliky.IN:= FALSE;
		doZatvorenieOdvzdHydrauliky:= FALSE;
		CasZapnutiaHydrauliky.IN:= TRUE;
	ELSE
		CasVypnutiaHydrauliky.IN:= TRUE;
		CasZapnutiaHydrauliky.IN:= FALSE;
	END_IF

	IF CasZapnutiaHydrauliky.Q THEN
		doHydraulika_ChodCerpadla:= TRUE;
	END_IF

	IF CasVypnutiaHydrauliky.Q THEN
		doZatvorenieOdvzdHydrauliky:= TRUE;
		doHydraulika_ChodCerpadla:= FALSE;
		Vyrazanie.OUT.VyrazanieZasunut:= FALSE;
		Vyrazanie.OUT.VyrazanieVysunut:= FALSE;
		doRazenie_ZostupRotora:= FALSE;
	END_IF

	CasZapnutiaHydrauliky.PT:= T#1s;
	CasZapnutiaHydrauliky();

	CasVypnutiaHydrauliky.PT:= T#60s;
	CasVypnutiaHydrauliky();

END_ACTION
```

### Program Logical/Program/Oddelovac (IEC)

#### Main.st - Init, cyclic, exit code
```iecst
PROGRAM _INIT
	(* Insert code here *)

END_PROGRAM

PROGRAM _CYCLIC

	//Volanie podprogramov//
	OvladanieOddelovaca;

	//Volanie funkcie SequenceControl//
	SequenceControl(SC:= SC_Oddelovac);

	//Reset sekcie //
	IF Oddelovac_Reset OR NOT BezpOkruhOplotenia_Aktivovany OR PoruchaOddelovaca THEN
		SC_Oddelovac.Step:= 0;
	END_IF

	CASE SC_Oddelovac.Step OF

		0:
			SC_Oddelovac.StepName:='0 - Nulovanie';
			SC_OvlOddelovaca.Step:= 0;
			Oddelovac_Automat:= FALSE;
			Oddelovac_KoniecVyroby:= FALSE;
			Oddelovac_KoniecCyklu:= FALSE;
			Oddelovac_Manual:= FALSE;
			Oddelovac_PoINIT:= FALSE;
			Oddelovac_Reset:= FALSE;
			IF BezpOkruhOplotenia_Aktivovany AND NOT PoruchaOddelovaca THEN
				SC_Oddelovac.ResetStep:= TRUE;
				SC_Oddelovac.Step:= 1;
			END_IF

		1:
			SC_Oddelovac.StepName:='1 - Rozhodnutie o cinnosti';
			IF Oddelovac_Automat THEN
				SC_Oddelovac.Step:= 2;
			ELSIF Oddelovac_Manual THEN
				SC_Oddelovac.Step:= 700;
			END_IF

		//********************************************************Inicializácia****************************************************************************//

		2:
			SC_Oddelovac.StepName:='2 - Inicializacia - cakanie na spustenie';
			SC_Oddelovac.IdleTime.PT:= T#500ms;
			SC_Oddelovac.AlarmTime.PT:= T#5s;
			SC_Oddelovac.IdleTime.IN:= TRUE;

			IF SC_Oddelovac.IdleTime.Q THEN
				SC_Oddelovac.ResetStep:= TRUE;
				SC_Oddelovac.Step:= 3;
			END_IF

		3:
			SC_Oddelovac.StepName:='3 - Inicializacia - rozhodnutie o preklopeni';
			SC_Oddelovac.IdleTime.PT:= T#500ms;
			SC_Oddelovac.AlarmTime.PT:= T#5s;

			IF NOT diOddelovac_PoziciaNavazanie AND NOT diOddelovac_PritomnostRotora THEN
				SC_Oddelovac.ResetStep:= TRUE;
				SC_Oddelovac.Step:= 4;
			ELSIF diOddelovac_PoziciaNavazanie THEN
				Oddelovac_PoINIT:= TRUE;
				SC_Oddelovac.ResetStep:= TRUE;
				SC_Oddelovac.Step:= 100;
			END_IF

		4:
			SC_Oddelovac.StepName:='4 - Inicializacia - preklopenie do navazacej pozicie';
			SC_Oddelovac.IdleTime.PT:= T#500ms;
			SC_Oddelovac.AlarmTime.PT:= T#5s;

			IF NOT SC_Oddelovac.Switch1 THEN
				Oddelovac_NAVAZANIE:= TRUE;
				SC_Oddelovac.Switch1:= TRUE;
			END_IF

			IF diOddelovac_PoziciaNavazanie THEN
				Oddelovac_PoINIT:= TRUE;
				SC_Oddelovac.ResetStep:= TRUE;
				SC_Oddelovac.Step:= 100;
			END_IF

		//********************************************************Automatický režim****************************************************************************//
		100:
			SC_Oddelovac.StepName:='100 - Automaticky rezim - cakanie na preklopenie do vyvazacej pozicie';
			SC_Oddelovac.IdleTime.PT:= T#500ms;
			SC_Oddelovac.AlarmTime.PT:= T#5s;

			IF diOddelovac_PritomnostRotora AND NOT diVstupDopr_PritomnostRotora AND (diVstupManipul_ZasunutyHore OR VstupManipulator_AktualPozMM < 600) AND NOT Oddelovac_KoniecVyroby AND diVstupDopr_ZdvihRotora_DOLE THEN
				SC_Oddelovac.IdleTime.IN:= TRUE;
			ELSE
				SC_Oddelovac.IdleTime.IN:= FALSE;
			END_IF

			IF SC_Oddelovac.IdleTime.Q THEN
				SC_Oddelovac.ResetStep:= TRUE;
				SC_Oddelovac.Step:= 101;
			END_IF

			IF Oddelovac_KoniecCyklu AND NOT VstupManipulator_Automat THEN
				SC_Oddelovac.ResetStep:= TRUE;
				SC_Oddelovac.Step:= 0;
			END_IF

			IF Oddelovac_KoniecVyroby AND NOT VstupManipulator_Automat THEN
				SC_Oddelovac.ResetStep:= TRUE;
				SC_Oddelovac.Step:= 0;
			END_IF

		101:
			SC_Oddelovac.StepName:='101 - Automaticky rezim - preklopenie do vyvazacej pozicie';
			SC_Oddelovac.IdleTime.PT:= T#500ms;
			SC_Oddelovac.AlarmTime.PT:= T#5s;

			IF NOT SC_Oddelovac.Switch1 THEN
				Oddelovac_VYVAZANIE:= TRUE;
				SC_Oddelovac.Switch1:= TRUE;
			END_IF

			IF diOddelovac_PoziciaVyvazanie THEN
				SC_Oddelovac.ResetStep:= TRUE;
				SC_Oddelovac.Step:= 102;
			END_IF

		102:
			SC_Oddelovac.StepName:='102 - Automaticky rezim - cakanie na preklopenie do navazacej pozicie';
			SC_Oddelovac.IdleTime.PT:= T#100ms;
			SC_Oddelovac.AlarmTime.PT:= T#5s;

			IF NOT diOddelovac_PritomnostRotora AND diVstupDopr_PritomnostRotora THEN
				SC_Oddelovac.IdleTime.IN:= TRUE;
			ELSE
				SC_Oddelovac.IdleTime.IN:= FALSE;
			END_IF

			IF SC_Oddelovac.IdleTime.Q THEN
				SC_Oddelovac.ResetStep:= TRUE;
				SC_Oddelovac.Step:= 103;
			END_IF

		103:
			SC_Oddelovac.StepName:='102 - Automaticky rezim - cakanie na preklopenie do navazacej pozicie';
			SC_Oddelovac.IdleTime.PT:= T#500ms;
			SC_Oddelovac.AlarmTime.PT:= T#5s;

			IF NOT SC_Oddelovac.Switch1 THEN
				Oddelovac_NAVAZANIE:= TRUE;
				SC_Oddelovac.Switch1:= TRUE;
			END_IF

			IF diOddelovac_PoziciaNavazanie THEN
				SC_Oddelovac.ResetStep:= TRUE;
				SC_Oddelovac.Step:= 100;
			END_IF

		//********************************************************Ručný režim***********************************************************************************//
		700:
			SC_Oddelovac.StepName:='700 - Rucny rezim';

	END_CASE

END_PROGRAM

PROGRAM _EXIT
	(* Insert code here *)

END_PROGRAM
```

#### Variables.var - Local variables
```iecst
VAR
	SC_OvlOddelovaca : SequenceControlTyp;
	Oddelovac_NAVAZANIE : BOOL;
	Oddelovac_VYVAZANIE : BOOL;
END_VAR
```

#### OvladanieOddelovaca.st
```iecst
ACTION OvladanieOddelovaca:

	//Volanie funkcie SequenceControl//
	SequenceControl(SC:= SC_OvlOddelovaca);

	CASE SC_OvlOddelovaca.Step OF

		0:
			SC_OvlOddelovaca.StepName:= '0 - Nulovanie';
			Oddelovac_NAVAZANIE:= FALSE;
			Oddelovac_VYVAZANIE:= FALSE;
			doOddelovac_PrepniPozNavazania:= FALSE;
			doOddelovac_PrepniPozVyvazania:= FALSE;
			IF SC_Oddelovac.Step <> 0 THEN
				SC_OvlOddelovaca.ResetStep:= TRUE;
				SC_OvlOddelovaca.Step:= 1;
			END_IF

		1:
			SC_OvlOddelovaca.StepName:= '1 - Rozhodnutie o cinnosti';
			IF Oddelovac_NAVAZANIE THEN
				SC_OvlOddelovaca.Step:= 10;
			ELSIF Oddelovac_VYVAZANIE THEN
				SC_OvlOddelovaca.Step:= 20;
			END_IF

		10:
			SC_OvlOddelovaca.StepName:= '10 - Prepnutie oddelovaca do polohy navazania';
			SC_OvlOddelovaca.IdleTime.PT:= T#3s;
			SC_OvlOddelovaca.AlarmTime.PT:= T#3s;
			IF Oddelovac_Manual THEN
				SC_OvlOddelovaca.IdleTime.IN:= TRUE;
			ELSE
				SC_OvlOddelovaca.AlarmTime.IN:= TRUE;
			END_IF

			IF NOT SC_OvlOddelovaca.Switch1 THEN
				doOddelovac_PrepniPozNavazania:= TRUE;
				SC_OvlOddelovaca.Switch1:= TRUE;
			END_IF

			IF SC_OvlOddelovaca.AlarmTime.Q THEN
				Alarmy[10]:= TRUE;
				PoruchaOddelovaca:= TRUE;
			END_IF

			IF (diOddelovac_PoziciaNavazanie AND NOT diOddelovac_PoziciaVyvazanie) OR SC_OvlOddelovaca.IdleTime.Q THEN
				SC_OvlOddelovaca.ResetStep:= TRUE;
				SC_OvlOddelovaca.Step:= 0;
			END_IF

		20:
			SC_OvlOddelovaca.StepName:= '20 - Prepnutie oddelovaca do polohy vyvazania';
			SC_OvlOddelovaca.IdleTime.PT:= T#3s;
			SC_OvlOddelovaca.AlarmTime.PT:= T#3s;
			IF Oddelovac_Manual THEN
				SC_OvlOddelovaca.IdleTime.IN:= TRUE;
			ELSE
				SC_OvlOddelovaca.AlarmTime.IN:= TRUE;
			END_IF

			IF NOT SC_OvlOddelovaca.Switch1 THEN
				doOddelovac_PrepniPozVyvazania:= TRUE;
				SC_OvlOddelovaca.Switch1:= TRUE;
			END_IF

			IF SC_OvlOddelovaca.AlarmTime.Q THEN
				Alarmy[10]:= TRUE;
				PoruchaOddelovaca:= TRUE;
			END_IF

			IF (diOddelovac_PoziciaVyvazanie AND NOT diOddelovac_PoziciaNavazanie) OR SC_OvlOddelovaca.IdleTime.Q THEN
				SC_OvlOddelovaca.ResetStep:= TRUE;
				SC_OvlOddelovaca.Step:= 0;
			END_IF

	END_CASE

END_ACTION
```

### Program Logical/Program/ZdvihRotora (IEC)

#### Main.st - Init, cyclic, exit code
```iecst
PROGRAM _INIT
	(* Insert code here *)

END_PROGRAM

PROGRAM _CYCLIC
	//Volanie podprogramov//
	OvladanieZdvihu;

	//Volanie funkcie SequenceControl//
	SequenceControl(SC:= SC_ZdvihRotora);

	//Reset sekcie //
	IF ZdvihRotora_Reset OR NOT BezpOkruhOplotenia_Aktivovany OR PoruchaZdvihuRotora THEN
		SC_ZdvihRotora.Step:= 0;
	END_IF

	CASE SC_ZdvihRotora.Step OF

		0:
			SC_ZdvihRotora.StepName:='0 - Nulovanie';
			SC_OvlZdvihu.Step:= 0;
			ZdvihRotora_Automat:= FALSE;
			ZdvihRotora_KoniecVyroby:= FALSE;
			ZdvihRotora_KoniecCyklu:= FALSE;
			ZdvihRotora_Manual:= FALSE;
			ZdvihRotora_PoINIT:= FALSE;
			ZdvihRotora_Reset:= FALSE;
			IF BezpOkruhOplotenia_Aktivovany AND NOT PoruchaZdvihuRotora THEN
				SC_ZdvihRotora.ResetStep:= TRUE;
				SC_ZdvihRotora.Step:= 1;
			END_IF

		1:
			SC_ZdvihRotora.StepName:='1 - Rozhodnutie o cinnosti';
			IF ZdvihRotora_Automat THEN
				SC_ZdvihRotora.Step:= 2;
			ELSIF ZdvihRotora_Manual THEN
				SC_ZdvihRotora.Step:= 700;
			END_IF

			//********************************************************Inicializácia****************************************************************************//

		2:
			SC_ZdvihRotora.StepName:='2 - Inicializacia - cakanie na spustenie';
			SC_ZdvihRotora.IdleTime.PT:= T#500ms;
			SC_ZdvihRotora.AlarmTime.PT:= T#5s;
			SC_ZdvihRotora.IdleTime.IN:= TRUE;

			IF SC_ZdvihRotora.IdleTime.Q THEN
				SC_ZdvihRotora.ResetStep:= TRUE;
				SC_ZdvihRotora.Step:= 3;
			END_IF

		3:
			SC_ZdvihRotora.StepName:='3 - Inicializacia - rozhodnutie o ukonceni inicializacie';
			SC_ZdvihRotora.IdleTime.PT:= T#500ms;
			SC_ZdvihRotora.AlarmTime.PT:= T#5s;

			IF diVstupDopr_ZdvihRotora_DOLE AND NOT diVstupDopr_ZdvihRotora_HORE THEN
				ZdvihRotora_PoINIT:= TRUE;
				SC_ZdvihRotora.ResetStep:= TRUE;
				SC_ZdvihRotora.Step:= 100;
			ELSIF diVstupDopr_ZdvihRotora_HORE AND NOT diVstupDopr_ZdvihRotora_DOLE AND diVstupDopr_PritomnostRotora THEN
				ZdvihRotora_PoINIT:= TRUE;
				SC_ZdvihRotora.ResetStep:= TRUE;
				SC_ZdvihRotora.Step:= 101;
			ELSIF diVstupDopr_ZdvihRotora_HORE AND NOT diVstupDopr_ZdvihRotora_DOLE AND NOT diVstupDopr_PritomnostRotora THEN
				SC_ZdvihRotora.ResetStep:= TRUE;
				SC_ZdvihRotora.Step:= 4;
			ELSE
				Alarmy[17]:= TRUE;
				PoruchaZdvihuRotora:= TRUE;
			END_IF

		4:
			SC_ZdvihRotora.StepName:='3 - Inicializacia - zasunutie zdvihu dole';
			SC_ZdvihRotora.IdleTime.PT:= T#500ms;
			SC_ZdvihRotora.AlarmTime.PT:= T#5s;

			IF NOT SC_ZdvihRotora.Switch1 THEN
				PolozRotor:= TRUE;
				SC_ZdvihRotora.Switch1:= TRUE;
			END_IF

			IF diVstupDopr_ZdvihRotora_DOLE THEN
				ZdvihRotora_PoINIT:= TRUE;
				SC_ZdvihRotora.ResetStep:= TRUE;
				SC_ZdvihRotora.Step:= 100;
			END_IF

			//********************************************************Automatický režim****************************************************************************//
		100:
			SC_ZdvihRotora.StepName:='100 - Automaticky rezim - cakanie na zdvihnutie rotora';
			SC_ZdvihRotora.IdleTime.PT:= T#200ms;
			SC_ZdvihRotora.AlarmTime.PT:= T#5s;

			IF diVstupDopr_PritomnostRotora THEN
				SC_ZdvihRotora.IdleTime.IN:= TRUE;
			ELSE
				SC_ZdvihRotora.IdleTime.IN:= FALSE;
			END_IF

			IF SC_ZdvihRotora.IdleTime.Q AND NOT SC_ZdvihRotora.Switch1 THEN
				ZdvihniRotor:= TRUE;
				SC_ZdvihRotora.Switch1:= TRUE;
			END_IF

			IF diVstupDopr_ZdvihRotora_HORE THEN
				SC_ZdvihRotora.ResetStep:= TRUE;
				SC_ZdvihRotora.Step:= 101;
			END_IF

			IF ZdvihRotora_KoniecCyklu AND NOT VstupManipulator_Automat THEN
				SC_ZdvihRotora.ResetStep:= TRUE;
				SC_ZdvihRotora.Step:= 0;
			END_IF

			IF ZdvihRotora_KoniecVyroby AND NOT VstupManipulator_Automat THEN
				SC_ZdvihRotora.ResetStep:= TRUE;
				SC_ZdvihRotora.Step:= 0;
			END_IF

		101:
			SC_ZdvihRotora.StepName:='101 - Automaticky rezim - cakanie na odobratie rotora';
			SC_ZdvihRotora.IdleTime.PT:= T#200ms;
			SC_ZdvihRotora.AlarmTime.PT:= T#5s;

			IF NOT diVstupDopr_PritomnostRotora THEN
				SC_ZdvihRotora.IdleTime.IN:= TRUE;
			ELSE
				SC_ZdvihRotora.IdleTime.IN:= FALSE;
			END_IF

			IF SC_ZdvihRotora.IdleTime.Q AND NOT SC_ZdvihRotora.Switch1 THEN
				PolozRotor:= TRUE;
				SC_ZdvihRotora.Switch1:= TRUE;
			END_IF

			IF diVstupDopr_ZdvihRotora_DOLE THEN
				SC_ZdvihRotora.ResetStep:= TRUE;
				SC_ZdvihRotora.Step:= 100;
			END_IF

			IF ZdvihRotora_KoniecCyklu AND NOT VstupManipulator_Automat THEN
				SC_ZdvihRotora.ResetStep:= TRUE;
				SC_ZdvihRotora.Step:= 0;
			END_IF

			IF ZdvihRotora_KoniecVyroby AND NOT VstupManipulator_Automat THEN
				SC_ZdvihRotora.ResetStep:= TRUE;
				SC_ZdvihRotora.Step:= 0;
			END_IF

			//********************************************************Ručný režim***********************************************************************************//
		700:
			SC_ZdvihRotora.StepName:='700 - Rucny rezim';

	END_CASE

				END_PROGRAM

PROGRAM _EXIT
				(* Insert code here *)

				END_PROGRAM
```

#### Variables.var - Local variables
```iecst
VAR
	SC_OvlZdvihu : SequenceControlTyp;
	ZdvihniRotor : BOOL;
	PolozRotor : BOOL;
END_VAR
```

#### OvladanieZdvihu.st
```iecst
ACTION OvladanieZdvihu:

	//Volanie funkcie SequenceControl//
	SequenceControl(SC:= SC_OvlZdvihu);

	CASE SC_OvlZdvihu.Step OF

		0:
			SC_OvlZdvihu.StepName:= '0 - Nulovanie';
			ZdvihniRotor:= FALSE;
			PolozRotor:= FALSE;
			IF SC_ZdvihRotora.Step <> 0 THEN
				SC_OvlZdvihu.ResetStep:= TRUE;
				SC_OvlZdvihu.Step:= 1;
			END_IF

		1:
			SC_OvlZdvihu.StepName:= '1 - Rozhodnutie o cinnosti';
			IF ZdvihniRotor THEN
				SC_OvlZdvihu.Step:= 10;
			ELSIF PolozRotor THEN
				SC_OvlZdvihu.Step:= 20;
			END_IF

		10:
			SC_OvlZdvihu.StepName:= '10 - Vysunutie zdvihu';
			SC_OvlZdvihu.IdleTime.PT:= T#1s;
			SC_OvlZdvihu.AlarmTime.PT:= T#3s;
			IF ZdvihRotora_Manual THEN
				SC_OvlZdvihu.IdleTime.IN:= TRUE;
			ELSE
				SC_OvlZdvihu.AlarmTime.IN:= TRUE;
			END_IF

			IF NOT SC_OvlZdvihu.Switch1 THEN
				doVstupDopr_VysunZdvihRotora:= TRUE;
				SC_OvlZdvihu.Switch1:= TRUE;
			END_IF

			IF SC_OvlZdvihu.AlarmTime.Q THEN
				Alarmy[15]:= TRUE;
				PoruchaZdvihuRotora:= TRUE;
			END_IF

			IF diVstupDopr_ZdvihRotora_HORE OR SC_OvlZdvihu.IdleTime.Q THEN
				SC_OvlZdvihu.ResetStep:= TRUE;
				SC_OvlZdvihu.Step:= 0;
			END_IF

		20:
			SC_OvlZdvihu.StepName:= '20 - Zasunutie zdvihu';
			SC_OvlZdvihu.IdleTime.PT:= T#1s;
			SC_OvlZdvihu.AlarmTime.PT:= T#3s;
			IF ZdvihRotora_Manual THEN
				SC_OvlZdvihu.IdleTime.IN:= TRUE;
			ELSE
				SC_OvlZdvihu.AlarmTime.IN:= TRUE;
			END_IF

			IF NOT SC_OvlZdvihu.Switch1 THEN
				doVstupDopr_VysunZdvihRotora:= FALSE;
				SC_OvlZdvihu.Switch1:= TRUE;
			END_IF

			IF SC_OvlZdvihu.AlarmTime.Q THEN
				Alarmy[16]:= TRUE;
				PoruchaZdvihuRotora:= TRUE;
			END_IF

			IF diVstupDopr_ZdvihRotora_DOLE OR SC_OvlZdvihu.IdleTime.Q THEN
				SC_OvlZdvihu.ResetStep:= TRUE;
				SC_OvlZdvihu.Step:= 0;
			END_IF

	END_CASE

END_ACTION
```

### Program Logical/Program/VstupnyManipulator (IEC)
